# B&R Automation Studio project TD52 (part 11)

#### Sim6CTR.c
```c
/********************************************************************
 * COPYRIGHT -- Bernecker + Rainer Industrie-Elektronik Ges.m.b.H.
 ********************************************************************
 * Program: Sim6CTR
 * File: Sim6CTR.c
 * Author: 105051472
 * Created: Wed Oct 23 10:19:46 2013
 ********************************************************************
 * Implementation of program Sim6CTR
 ********************************************************************
 * Generated with B&R Automation Studio Target for Simulink V4.0
 * (ERT based)
 ********************************************************************/
#include "Sim6CTR.h"
#include "Sim6CTR_private.h"

/*  Defines */

/* Named constants for Chart: '<S1>/Chart' */
#define Sim6CTR_IN_Close_CBP_3u4       ((uint8_T)1U)
#define Sim6CTR_IN_LoadDrop            ((uint8_T)1U)
#define Sim6CTR_IN_Lock_TV             ((uint8_T)1U)
#define Sim6CTR_IN_NO_ACTIVE_CHILD     ((uint8_T)0U)
#define Sim6CTR_IN_Open_CBP_3u4        ((uint8_T)2U)
#define Sim6CTR_IN_Release_TV          ((uint8_T)2U)
#define Sim6CTR_IN_Standard            ((uint8_T)2U)

/*  Data Types */

/**************************** GLOBAL DATA *************************************/
/*  Definitions */

/* Block signals (auto storage) */

/* Block states (auto storage) */

/*  Declarations  */

/***************************** FILE SCOPE DATA ********************************/

/*************************** FUNCTIONS ****************************************/

/* Model step function */
void Sim6CTR_step(struct Sim6CTR* inst)
{
  real_T rtb_Product;
  real_T rtb_Trackingswitch;
  real32_T rtb_Product2_g;
  real32_T rtb_Product1;
  real32_T rtb_Product2_b;
  real32_T rtb_Sum;
  real32_T rtb_Saturation;
  int32_T rtb_Switch1;
  real32_T rtb_Switch_h;
  boolean_T rtb_RelationalOperator2;
  real32_T rtb_Abs;
  real32_T rtb_SumI1;
  real32_T rtb_Saturation_o;
  real32_T rtb_Switch2;
  boolean_T rtb_Compare_e;

  /* S-Function (bur_in): '<Root>/Input10' */
  inst->bur_Sim6CTR_B.Input10 = inst->bInit;

  /* Switch: '<S1>/Switch1' incorporates:
   *  Constant: '<S1>/Constant12'
   *  Constant: '<S1>/Constant3'
   */
  if (inst->bur_Sim6CTR_B.Input10) {
    rtb_Switch1 = 2;
  } else {
    rtb_Switch1 = 3;
  }

  /* End of Switch: '<S1>/Switch1' */

  /* S-Function (bur_in): '<Root>/Input11' */
  inst->bur_Sim6CTR_B.Input11 = inst->Init_Value_CBP;

  /* S-Function (bur_in): '<Root>/Input1' */
  inst->bur_Sim6CTR_B.Input1 = inst->w_set;

  /* Product: '<S7>/Product' */
  rtb_Product = inst->bur_Sim6CTR_B.Input1;

  /* S-Function (bur_in): '<Root>/Input9' */
  inst->bur_Sim6CTR_B.Input9 = inst->x_act;

  /* Sum: '<S7>/Sum' incorporates:
   *  Product: '<S7>/Product1'
   */
  rtb_Product -= (real_T)inst->bur_Sim6CTR_B.Input9;

  /* DeadZone: '<S7>/Deadband' */
  if ((!(rtb_Product > 0.0)) && (rtb_Product >= -0.0)) {
    rtb_Product = 0.0;
  }

  /* End of DeadZone: '<S7>/Deadband' */

  /* Product: '<S7>/Product2' */
  rtb_Product2_g = (real32_T)-rtb_Product;

  /* S-Function (bur_in): '<Root>/Input3' */
  inst->bur_Sim6CTR_B.Input3 = inst->P_CBP;

  /* Product: '<S10>/Product1' incorporates:
   *  Product: '<S7>/Product2'
   */
  rtb_Product1 = (real32_T)-rtb_Product * inst->bur_Sim6CTR_B.Input3;

  /* DiscreteIntegrator: '<S10>/Integrator' */
  rtb_Product2_b = inst->bur_Sim6CTR_DWork.Integrator_DSTATE;

  /* S-Function (bur_in): '<Root>/Input5' */
  inst->bur_Sim6CTR_B.Input5 = inst->D_CBP;

  /* Sum: '<S10>/Sum2' incorporates:
   *  Sum: '<S10>/Sum1'
   */
  rtb_Sum = rtb_Product1 + rtb_Product2_b;

  /* Saturate: '<S10>/Saturation' */
  if (rtb_Sum >= inst->u_max_CBP) {
    rtb_Saturation = inst->u_max_CBP;
  } else if (rtb_Sum <= inst->u_min_CBP) {
    rtb_Saturation = inst->u_min_CBP;
  } else {
    rtb_Saturation = rtb_Sum;
  }

  /* End of Saturate: '<S10>/Saturation' */

  /* MultiPortSwitch: '<S7>/Mode switch' */
  switch (rtb_Switch1) {
   case 1:
    inst->bur_Sim6CTR_B.Modeswitch = inst->bur_Sim6CTR_B.Input11;
    break;

   case 2:
    inst->bur_Sim6CTR_B.Modeswitch = inst->bur_Sim6CTR_B.Input11;
    break;

   default:
    inst->bur_Sim6CTR_B.Modeswitch = rtb_Saturation;
    break;
  }

  /* End of MultiPortSwitch: '<S7>/Mode switch' */

  /* S-Function (bur_out): '<Root>/Output' */
  inst->rPos_CBP = inst->bur_Sim6CTR_B.Modeswitch;

  /* S-Function (bur_in): '<Root>/Input13' */
  inst->bur_Sim6CTR_B.Input13 = inst->rN_act;

  /* S-Function (bur_in): '<Root>/Input12' */
  inst->bur_Sim6CTR_B.Input12 = inst->rN_set;

  /* RelationalOperator: '<S1>/Relational Operator1' incorporates:
   *  Constant: '<S1>/rN_ok_offset'
   *  Sum: '<S1>/Add'
   */
  inst->bur_Sim6CTR_B.RelationalOperator1 = (inst->bur_Sim6CTR_B.Input13 < inst->bur_Sim6CTR_B.Input12 +
    inst->rN_ok_offset);

  /* Switch: '<S9>/Switch' incorporates:
   *  Constant: '<S1>/Cyclic Time'
   *  Constant: '<S9>/Constant4'
   *  Sum: '<S9>/Add'
   *  UnitDelay: '<S6>/Unit Delay2'
   *  UnitDelay: '<S9>/Unit Delay'
   */
  if (inst->bur_Sim6CTR_DWork.UnitDelay2_DSTATE) {
    rtb_Switch_h = 0.0F;
  } else {
    rtb_Switch_h = (real32_T)((real_T)inst->CycleTime + (real_T)
      inst->bur_Sim6CTR_DWork.UnitDelay_DSTATE);
  }

  /* End of Switch: '<S9>/Switch' */

  /* RelationalOperator: '<S6>/Relational Operator2' incorporates:
   *  Constant: '<S1>/Ts_downSampling_speed'
   */
  rtb_RelationalOperator2 = (rtb_Switch_h >= inst->Ts_downSampling_speed);

  /* Switch: '<S6>/Switch' incorporates:
   *  UnitDelay: '<S6>/Unit Delay'
   */
  if (rtb_RelationalOperator2) {
    inst->bur_Sim6CTR_B.Switch = inst->bur_Sim6CTR_B.Input13;
  } else {
    inst->bur_Sim6CTR_B.Switch = inst->bur_Sim6CTR_DWork.UnitDelay_DSTATE_e;
  }

  /* End of Switch: '<S6>/Switch' */

  /* Sum: '<S5>/Diff' incorporates:
   *  UnitDelay: '<S5>/UD'
   */
  inst->bur_Sim6CTR_B.Diff = inst->bur_Sim6CTR_B.Switch - inst->bur_Sim6CTR_DWork.UD_DSTATE;

  /* RelationalOperator: '<S4>/Compare' incorporates:
   *  Constant: '<S4>/Constant'
   */
  inst->bur_Sim6CTR_B.Compare = (inst->bur_Sim6CTR_B.Diff < 0.0F);

  /* Delay: '<S1>/Delay' */
  rtb_Product1 = inst->bur_Sim6CTR_DWork.Delay_DSTATE[0];

  /* S-Function (bur_in): '<Root>/Input2' */
  inst->bur_Sim6CTR_B.Input2 = inst->rP_el;

  /* Sum: '<S1>/Add1' */
  inst->bur_Sim6CTR_B.Add1 = inst->bur_Sim6CTR_B.Input2 - rtb_Product1;

  /* RelationalOperator: '<S1>/Relational Operator' incorporates:
   *  Constant: '<S1>/rP_drop_limit'
   */
  inst->bur_Sim6CTR_B.RelationalOperator = (inst->bur_Sim6CTR_B.Add1 < inst->rP_drop_limit);

  /* Chart: '<S1>/Chart' incorporates:
   *  Constant: '<S1>/rP_el_LockTV'
   *  MinMax: '<S1>/MinMax'
   *  UnitDelay: '<S1>/Unit Delay'
   */
  /* Gateway: Island Controller/Chart */
  /* During: Island Controller/Chart */
  if (inst->bur_Sim6CTR_DWork.is_active_c1_Sim6CTR == 0U) {
    /* Entry: Island Controller/Chart */
    inst->bur_Sim6CTR_DWork.is_active_c1_Sim6CTR = 1U;

    /* Entry Internal: Island Controller/Chart */
    /* Transition: '<S3>:12' */
    inst->bur_Sim6CTR_DWork.is_c1_Sim6CTR = Sim6CTR_IN_Standard;

    /* Entry 'Standard': '<S3>:7' */
    inst->bur_Sim6CTR_B.bLoadDrop = FALSE;
    inst->bur_Sim6CTR_B.Open4CBP = FALSE;

    /* Entry Internal 'Standard': '<S3>:7' */
    /* Transition: '<S3>:16' */
    inst->bur_Sim6CTR_DWork.is_Standard = Sim6CTR_IN_Release_TV;

    /* Entry 'Release_TV': '<S3>:15' */
    inst->bur_Sim6CTR_B.Lock_TV = FALSE;
    inst->bur_Sim6CTR_B.Control_State = 11;
  } else if (inst->bur_Sim6CTR_DWork.is_c1_Sim6CTR == Sim6CTR_IN_LoadDrop) {
    /* During 'LoadDrop': '<S3>:10' */
    if (inst->bur_Sim6CTR_B.RelationalOperator1 && inst->bur_Sim6CTR_B.Compare) {
      /* Transition: '<S3>:25' */
      /* Exit Internal 'LoadDrop': '<S3>:10' */
      inst->bur_Sim6CTR_DWork.is_LoadDrop = Sim6CTR_IN_NO_ACTIVE_CHILD;
      inst->bur_Sim6CTR_DWork.is_c1_Sim6CTR = Sim6CTR_IN_Standard;

      /* Entry 'Standard': '<S3>:7' */
      inst->bur_Sim6CTR_B.bLoadDrop = FALSE;
      inst->bur_Sim6CTR_B.Open4CBP = FALSE;

      /* Entry Internal 'Standard': '<S3>:7' */
      /* Transition: '<S3>:16' */
      inst->bur_Sim6CTR_DWork.is_Standard = Sim6CTR_IN_Release_TV;

      /* Entry 'Release_TV': '<S3>:15' */
      inst->bur_Sim6CTR_B.Lock_TV = FALSE;
      inst->bur_Sim6CTR_B.Control_State = 11;
    } else {
      switch (inst->bur_Sim6CTR_DWork.is_LoadDrop) {
       case Sim6CTR_IN_Close_CBP_3u4:
        break;

       default:
        /* During 'Open_CBP_3u4': '<S3>:29' */
        if (inst->bur_Sim6CTR_B.Compare) {
          /* Transition: '<S3>:32' */
          inst->bur_Sim6CTR_DWork.is_LoadDrop = Sim6CTR_IN_Close_CBP_3u4;

          /* Entry 'Close_CBP_3u4': '<S3>:31' */
          inst->bur_Sim6CTR_B.Open4CBP = FALSE;
          inst->bur_Sim6CTR_B.Control_State = 22;
        }
        break;
      }
    }
  } else {
    /* During 'Standard': '<S3>:7' */
    if (inst->bur_Sim6CTR_B.RelationalOperator) {
      /* Transition: '<S3>:23' */
      /* Exit Internal 'Standard': '<S3>:7' */
      inst->bur_Sim6CTR_DWork.is_Standard = Sim6CTR_IN_NO_ACTIVE_CHILD;
      inst->bur_Sim6CTR_DWork.is_c1_Sim6CTR = Sim6CTR_IN_LoadDrop;

      /* Entry 'LoadDrop': '<S3>:10' */
      inst->bur_Sim6CTR_B.Lock_TV = FALSE;
      inst->bur_Sim6CTR_B.bLoadDrop = TRUE;

      /* Entry Internal 'LoadDrop': '<S3>:10' */
      /* Transition: '<S3>:30' */
      inst->bur_Sim6CTR_DWork.is_LoadDrop = Sim6CTR_IN_Open_CBP_3u4;

      /* Entry 'Open_CBP_3u4': '<S3>:29' */
      inst->bur_Sim6CTR_B.Open4CBP = TRUE;
      inst->bur_Sim6CTR_B.Control_State = 21;
    } else if (inst->bur_Sim6CTR_DWork.is_Standard == Sim6CTR_IN_Lock_TV) {
      /* MinMax: '<S1>/MinMax' incorporates:
       *  Constant: '<S1>/rP_el_LockTV'
       *  Constant: '<S1>/rP_el_ReleaseTV'
       */
      /* During 'Lock_TV': '<S3>:9' */
      if (inst->rP_el_LockTV <= inst->rP_el_ReleaseTV) {
        rtb_Product = inst->rP_el_LockTV;
      } else {
        rtb_Product = inst->rP_el_ReleaseTV;
      }

      if ((real_T)inst->bur_Sim6CTR_B.Input2 < rtb_Product) {
        /* Transition: '<S3>:20' */
        inst->bur_Sim6CTR_DWork.is_Standard = Sim6CTR_IN_Release_TV;

        /* Entry 'Release_TV': '<S3>:15' */
        inst->bur_Sim6CTR_B.Lock_TV = FALSE;
        inst->bur_Sim6CTR_B.Control_State = 11;
      }
    } else {
      /* During 'Release_TV': '<S3>:15' */
      if ((inst->bur_Sim6CTR_B.Input2 > inst->rP_el_LockTV) && (inst->bur_Sim6CTR_DWork.UnitDelay_DSTATE_n
           > 72.0F)) {
        /* Transition: '<S3>:19' */
        inst->bur_Sim6CTR_DWork.is_Standard = Sim6CTR_IN_Lock_TV;

        /* Entry 'Lock_TV': '<S3>:9' */
        inst->bur_Sim6CTR_B.Lock_TV = TRUE;
        inst->bur_Sim6CTR_B.Control_State = 12;
      }
    }
  }

  /* End of Chart: '<S1>/Chart' */

  /* Switch: '<S1>/Switch' incorporates:
   *  Constant: '<S1>/Constant2'
   *  Constant: '<S1>/Constant31'
   *  Logic: '<S1>/Logical Operator'
   */
  if (inst->bur_Sim6CTR_B.Input10 || inst->bur_Sim6CTR_B.Lock_TV) {
    rtb_Product = 2.0;
  } else {
    rtb_Product = 3.0;
  }

  /* End of Switch: '<S1>/Switch' */

  /* S-Function (bur_in): '<Root>/Input14' */
  inst->bur_Sim6CTR_B.Input14 = inst->Init_Value_TV;

  /* Switch: '<S1>/Switch2' incorporates:
   *  Constant: '<S1>/u_man_TV'
   */
  if (inst->bur_Sim6CTR_B.Input10) {
    rtb_Switch2 = inst->bur_Sim6CTR_B.Input14;
  } else {
    rtb_Switch2 = inst->u_man_TV;
  }

  /* End of Switch: '<S1>/Switch2' */

  /* Sum: '<S8>/Sum' incorporates:
   *  Product: '<S8>/Product'
   *  Product: '<S8>/Product1'
   */
  rtb_Trackingswitch = (real_T)inst->bur_Sim6CTR_B.Input1 - (real_T)inst->bur_Sim6CTR_B.Input9;

  /* DeadZone: '<S8>/Deadband' */
  if ((!(rtb_Trackingswitch > 0.0)) && (rtb_Trackingswitch >= -0.0)) {
    rtb_Trackingswitch = 0.0;
  }

  /* End of DeadZone: '<S8>/Deadband' */

  /* Product: '<S8>/Product2' */
  rtb_Product2_b = (real32_T)rtb_Trackingswitch;

  /* S-Function (bur_in): '<Root>/Input6' */
  inst->bur_Sim6CTR_B.Input6 = inst->P_TV;

  /* Product: '<S13>/Product1' incorporates:
   *  Product: '<S8>/Product2'
   */
  rtb_Product1 = (real32_T)rtb_Trackingswitch * inst->bur_Sim6CTR_B.Input6;

  /* DiscreteIntegrator: '<S13>/Integrator' */
  rtb_Abs = inst->bur_Sim6CTR_DWork.Integrator_DSTATE_i;

  /* S-Function (bur_in): '<Root>/Input8' */
  inst->bur_Sim6CTR_B.Input8 = inst->D_TV;

  /* Sum: '<S13>/Sum2' incorporates:
   *  Sum: '<S13>/Sum1'
   */
  rtb_SumI1 = rtb_Product1 + rtb_Abs;

  /* Saturate: '<S13>/Saturation' */
  if (rtb_SumI1 >= inst->u_max_TV) {
    rtb_Saturation_o = inst->u_max_TV;
  } else if (rtb_SumI1 <= inst->u_min_TV) {
    rtb_Saturation_o = inst->u_min_TV;
  } else {
    rtb_Saturation_o = rtb_SumI1;
  }

  /* End of Saturate: '<S13>/Saturation' */

  /* MultiPortSwitch: '<S8>/Mode switch' */
  switch ((int32_T)rtb_Product) {
   case 1:
    inst->bur_Sim6CTR_B.Modeswitch_a = rtb_Switch2;
    break;

   case 2:
    inst->bur_Sim6CTR_B.Modeswitch_a = rtb_Switch2;
    break;

   default:
    inst->bur_Sim6CTR_B.Modeswitch_a = rtb_Saturation_o;
    break;
  }

  /* End of MultiPortSwitch: '<S8>/Mode switch' */

  /* S-Function (bur_out): '<Root>/Output1' */
  inst->rPos_TV = inst->bur_Sim6CTR_B.Modeswitch_a;

  /* S-Function (bur_out): '<Root>/Output10' */
  inst->rN_act_Diff = inst->bur_Sim6CTR_B.Diff;

  /* S-Function (bur_out): '<Root>/Output11' */
  inst->bOpen4CBP = inst->bur_Sim6CTR_B.Open4CBP;

  /* S-Function (bur_out): '<Root>/Output2' */
  inst->bLoadDrop = inst->bur_Sim6CTR_B.bLoadDrop;

  /* S-Function (bur_out): '<Root>/Output3' */
  inst->Control_State = inst->bur_Sim6CTR_B.Control_State;

  /* S-Function (bur_out): '<Root>/Output4' */
  inst->bLock_TV = inst->bur_Sim6CTR_B.Lock_TV;

  /* S-Function (bur_out): '<Root>/Output5' */
  inst->bN_ok = inst->bur_Sim6CTR_B.RelationalOperator1;

  /* S-Function (bur_out): '<Root>/Output6' */
  inst->bN_rate_neg = inst->bur_Sim6CTR_B.Compare;

  /* S-Function (bur_out): '<Root>/Output7' */
  inst->bP_drop = inst->bur_Sim6CTR_B.RelationalOperator;

  /* S-Function (bur_out): '<Root>/Output8' */
  inst->rP_grad = inst->bur_Sim6CTR_B.Add1;

  /* S-Function (bur_out): '<Root>/Output9' */
  inst->rN_act_DS = inst->bur_Sim6CTR_B.Switch;

  /* S-Function (bur_in): '<Root>/Input4' */
  inst->bur_Sim6CTR_B.Input4 = inst->I_CBP;

  /* S-Function (bur_in): '<Root>/Input7' */
  inst->bur_Sim6CTR_B.Input7 = inst->I_TV;

  /* Sum: '<S11>/Sum' */
  rtb_Sum = rtb_Saturation - rtb_Sum;

  /* MultiPortSwitch: '<S7>/Tracking switch' incorporates:
   *  Constant: '<S7>/Constant'
   *  Constant: '<S7>/Constant1'
   */
  switch (rtb_Switch1) {
   case 1:
    rtb_Trackingswitch = 0.0;
    break;

   case 2:
    rtb_Trackingswitch = 1.0;
    break;

   default:
    rtb_Trackingswitch = 0.0;
    break;
  }

  /* End of MultiPortSwitch: '<S7>/Tracking switch' */

  /* Sum: '<S10>/SumI1' incorporates:
   *  Product: '<S10>/Product'
   *  Product: '<S10>/Product2'
   *  Sum: '<S10>/SumI3'
   */
  rtb_Abs = (real32_T)((real_T)(inst->bur_Sim6CTR_B.Input11 - rtb_Saturation) *
                       rtb_Trackingswitch) + rtb_Product2_g * inst->bur_Sim6CTR_B.Input4;

  /* Signum: '<S11>/SignPreSat' */
  if (rtb_Sum < 0.0F) {
    rtb_Product2_g = -1.0F;
  } else if (rtb_Sum > 0.0F) {
    rtb_Product2_g = 1.0F;
  } else {
    rtb_Product2_g = rtb_Sum;
  }

  /* Signum: '<S11>/SignPreIntegrator' */
  if (rtb_Abs < 0.0F) {
    rtb_Saturation = -1.0F;
  } else if (rtb_Abs > 0.0F) {
    rtb_Saturation = 1.0F;
  } else {
    rtb_Saturation = rtb_Abs;
  }

  /* Switch: '<S10>/Switch' incorporates:
   *  Abs: '<S11>/Abs'
   *  Constant: '<S10>/Constant4'
   *  Constant: '<S12>/Constant'
   *  Logic: '<S11>/AND'
   *  RelationalOperator: '<S11>/Equal'
   *  RelationalOperator: '<S12>/Compare'
   *  Signum: '<S11>/SignPreIntegrator'
   *  Signum: '<S11>/SignPreSat'
   */
  if (((real32_T)fabs(rtb_Sum) > 0.1F) && (rtb_Product2_g != rtb_Saturation)) {
    rtb_Abs = 0.0F;
  }

  /* End of Switch: '<S10>/Switch' */

  /* Sum: '<S14>/Sum' */
  rtb_SumI1 = rtb_Saturation_o - rtb_SumI1;

  /* RelationalOperator: '<S15>/Compare' incorporates:
   *  Abs: '<S14>/Abs'
   *  Constant: '<S15>/Constant'
   */
  rtb_Compare_e = ((real32_T)fabs(rtb_SumI1) > 0.1F);

  /* Signum: '<S14>/SignPreSat' */
  if (rtb_SumI1 < 0.0F) {
    rtb_Product1 = -1.0F;
  } else if (rtb_SumI1 > 0.0F) {
    rtb_Product1 = 1.0F;
  } else {
    rtb_Product1 = rtb_SumI1;
  }

  /* End of Signum: '<S14>/SignPreSat' */

  /* MultiPortSwitch: '<S8>/Tracking switch' incorporates:
   *  Constant: '<S8>/Constant'
   *  Constant: '<S8>/Constant1'
   */
  switch ((int32_T)rtb_Product) {
   case 1:
    rtb_Trackingswitch = 0.0;
    break;

   case 2:
    rtb_Trackingswitch = 1.0;
    break;

   default:
    rtb_Trackingswitch = 0.0;
    break;
  }

  /* End of MultiPortSwitch: '<S8>/Tracking switch' */

  /* Sum: '<S13>/SumI1' incorporates:
   *  Product: '<S13>/Product'
   *  Product: '<S13>/Product2'
   *  Sum: '<S13>/SumI3'
   */
  rtb_SumI1 = (real32_T)((real_T)(rtb_Switch2 - rtb_Saturation_o) *
    rtb_Trackingswitch) + rtb_Product2_b * inst->bur_Sim6CTR_B.Input7;

  /* Signum: '<S14>/SignPreIntegrator' */
  if (rtb_SumI1 < 0.0F) {
    rtb_Product2_g = -1.0F;
  } else if (rtb_SumI1 > 0.0F) {
    rtb_Product2_g = 1.0F;
  } else {
    rtb_Product2_g = rtb_SumI1;
  }

  /* Switch: '<S13>/Switch' incorporates:
   *  Constant: '<S13>/Constant4'
   *  Logic: '<S14>/AND'
   *  RelationalOperator: '<S14>/Equal'
   *  Signum: '<S14>/SignPreIntegrator'
   */
  if (rtb_Compare_e && (rtb_Product1 != rtb_Product2_g)) {
    rtb_Product1 = 0.0F;
  } else {
    rtb_Product1 = rtb_SumI1;
  }

  /* End of Switch: '<S13>/Switch' */

  /* Update for DiscreteIntegrator: '<S10>/Integrator' */
  inst->bur_Sim6CTR_DWork.Integrator_DSTATE += 0.01F * rtb_Abs;

  /* Update for UnitDelay: '<S6>/Unit Delay2' */
  inst->bur_Sim6CTR_DWork.UnitDelay2_DSTATE = rtb_RelationalOperator2;

  /* Update for UnitDelay: '<S9>/Unit Delay' */
  inst->bur_Sim6CTR_DWork.UnitDelay_DSTATE = rtb_Switch_h;

  /* Update for UnitDelay: '<S6>/Unit Delay' */
  inst->bur_Sim6CTR_DWork.UnitDelay_DSTATE_e = inst->bur_Sim6CTR_B.Switch;

  /* Update for UnitDelay: '<S5>/UD' */
  inst->bur_Sim6CTR_DWork.UD_DSTATE = inst->bur_Sim6CTR_B.Switch;

  /* Update for Delay: '<S1>/Delay' */
  for (rtb_Switch1 = 0; rtb_Switch1 < 9; rtb_Switch1++) {
    inst->bur_Sim6CTR_DWork.Delay_DSTATE[rtb_Switch1] =
      inst->bur_Sim6CTR_DWork.Delay_DSTATE[rtb_Switch1 + 1];
  }

  inst->bur_Sim6CTR_DWork.Delay_DSTATE[9] = inst->bur_Sim6CTR_B.Input2;

  /* End of Update for Delay: '<S1>/Delay' */

  /* Update for UnitDelay: '<S1>/Unit Delay' */
  inst->bur_Sim6CTR_DWork.UnitDelay_DSTATE_n = inst->bur_Sim6CTR_B.Modeswitch_a;

  /* Update for DiscreteIntegrator: '<S13>/Integrator' */
  inst->bur_Sim6CTR_DWork.Integrator_DSTATE_i += 0.01F * rtb_Product1;
}

/* Model initialize function */
void Sim6CTR_initialize(struct Sim6CTR* inst)
{
  /* InitializeConditions for Chart: '<S1>/Chart' */
  inst->bur_Sim6CTR_B.Control_State = 0;
  inst->bur_Sim6CTR_B.Lock_TV = FALSE;
  inst->bur_Sim6CTR_B.bLoadDrop = FALSE;
  inst->bur_Sim6CTR_B.Open4CBP = FALSE;
}

/* Model terminate function */
void Sim6CTR_terminate(struct Sim6CTR* inst)
{
  /* (no terminate code required) */
}

/*======================== TOOL VERSION INFORMATION ==========================*
 * MATLAB 8.0 (R2012b)20-Jul-2012                                             *
 * Simulink 8.0 (R2012b)20-Jul-2012                                           *
 * Simulink Coder 8.3 (R2012b)20-Jul-2012                                     *
 * Embedded Coder 6.3 (R2012b)20-Jul-2012                                     *
 * Stateflow 8.0 (R2012b)20-Jul-2012                                          *
 *============================================================================*/

/*======================= LICENSE IN USE INFORMATION =========================*
 * control_toolbox                                                            *
 * identification_toolbox                                                     *
 * matlab                                                                     *
 * matlab_coder                                                               *
 * real-time_workshop                                                         *
 * rtw_embedded_coder                                                         *
 * simulink                                                                   *
 * stateflow                                                                  *
 *============================================================================*/
```

#### main.c
```c
/********************************************************************
 * COPYRIGHT -- Bernecker + Rainer Industrie-Elektronik Ges.m.b.H.
 ********************************************************************
 * Program: Sim6CTR
 * File: main.c
 * Author: 105051472
 * Created: Wed Oct 23 10:19:46 2013
 ********************************************************************
 * Implementation of program Sim6CTR
 ********************************************************************
 * Generated with B&R Automation Studio Target for Simulink V4.0
 * (ERT based)
 ********************************************************************/
#include <bur/plctypes.h>
#include "Sim6CTR.h"
#include "rtwtypes.h"

BOOL bur_firsttime = TRUE;

/*  Defines */
#define SS_TERMINATE 4
#define SS_OUTPUT 3
#define SS_INITIALIZE 2

/*  Data Types */

/**************************** GLOBAL DATA *************************************/
/*  Definitions */

/*  Declarations  */

/***************************** FILE SCOPE DATA ********************************/

/*************************** FUNCTIONS ****************************************/
#ifdef __cplusplus

unsigned long bur_heap_size = 65535;

#endif

void Sim6CTR(struct Sim6CTR* inst)
{
  switch (inst->ssMethodType)
  {
   case SS_INITIALIZE:
    /* call model initialize function */
    Sim6CTR_initialize(inst);
    break;

   case SS_OUTPUT:
    /* call model step function */
    Sim6CTR_step(inst);

    break;

   case SS_TERMINATE:
    /* call model terminate function */
    Sim6CTR_terminate(inst);
    break;
  }
}

/*****************************************************************************
   Function block sample time: 0.01s
 *****************************************************************************/

/*****************************************************************************
   B&R Automation Studio Target for Simulink Version: A4.0.48 (27-Jun-2013)
 *****************************************************************************/

/*======================== TOOL VERSION INFORMATION ==========================*
 * MATLAB 8.0 (R2012b)20-Jul-2012                                             *
 * Simulink 8.0 (R2012b)20-Jul-2012                                           *
 * Simulink Coder 8.3 (R2012b)20-Jul-2012                                     *
 * Embedded Coder 6.3 (R2012b)20-Jul-2012                                     *
 * Stateflow 8.0 (R2012b)20-Jul-2012                                          *
 *============================================================================*/

/*======================= LICENSE IN USE INFORMATION =========================*
 * control_toolbox                                                            *
 * identification_toolbox                                                     *
 * matlab                                                                     *
 * matlab_coder                                                               *
 * real-time_workshop                                                         *
 * rtw_embedded_coder                                                         *
 * simulink                                                                   *
 * stateflow                                                                  *
 *============================================================================*/
```

#### lib_properties.txt
```
For manual assignment to hardware configuration please
add the following additional include directories:

\Logical\MATLAB_includes\R2012b\

And the following additional build options:

-lm -D MODEL=Sim6CTR -D NUMST=1 -D NCSTATES=0 -D HAVESTDIO -D ONESTEPFCN=1 -D TERMFCN=1 -D MAT_FILE=0 -D MULTI_INSTANCE_CODE=0 -D INTEGER_CODE=0 -D MT=0 -D CLASSIC_INTERFACE=0 -D TID01EQ=0
```

### Library Logical/Libraries/lLamCorr (ANSIC)

#### lLamCorr.fun
```iecst
FUNCTION_BLOCK lLamCorr
  VAR_INPUT
    ssMethodType: SINT;
  END_VAR  VAR_INPUT
        rN_Set : REAL := 1500.0000000000; (*speed set value [rpm]*)
  END_VAR
  VAR_INPUT
        rP_Nom : REAL := 4400.0000000000; (*nominal power [KW]*)
  END_VAR
  VAR_INPUT
        rN_Delta_Lim : REAL := 0.0099999998; (*delta speed limit when engine speed is recovered, normed*)
  END_VAR
  VAR_INPUT
        rP_Rot_Norm_Lam_Trig : REAL := 0.0199999996; (*rotational power trigger value for lambda adaption, normed*)
  END_VAR
  VAR_INPUT
        rP_Rot_Norm_Lambda_Gain : REAL := 1.0000000000; (*gain value to convert nomed rotational power to delta lambda value for lambda adaption*)
  END_VAR
  VAR_INPUT
        rLam_OffsLimit_pos : REAL; (*pos limitation of dynamic lambda offset*)
  END_VAR
  VAR_INPUT
        rLam_Ramp_Grad : REAL := 0.2500000000; (*neg limitation of dynamic lambda offset*)
  END_VAR
  VAR_INPUT
        bLambda_Corr_Enable : BOOL := FALSE; (*enable function of lambda correction*)
  END_VAR
  VAR_INPUT
        rP_Rot : REAL; (*rotational power*)
  END_VAR
  VAR_INPUT
        rN_Eng : REAL; (*engine speed [rpm]*)
  END_VAR
  VAR_INPUT
        rLam_OffsLimit_Neg : REAL; (*engine speed [rpm]*)
  END_VAR
  VAR_OUTPUT
        rLambda_Corr : REAL; (*Lambda adaption value*)
  END_VAR
  VAR_OUTPUT
        bLambda_Freeze : BOOL := FALSE; (*Lambda adaption value*)
  END_VAR
  VAR_OUTPUT
        rP_Rot_Max : REAL; (*maximum value for rotational power, used for calibration*)
  END_VAR
  VAR_OUTPUT
        bN_Delta_Act : BOOL := FALSE; (*Debug Output*)
  END_VAR
  VAR_OUTPUT
        bP_Rot_Lambda_Act : BOOL := FALSE; (*Debug Output*)
  END_VAR
  VAR_OUTPUT
        bN_Delta_Neg : BOOL := FALSE; (*Debug Output*)
  END_VAR
	VAR
		bur_BlockIO_LambdaAdp : BlockIO_LambdaAdp;
	END_VAR
	VAR
		bur_D_Work_LambdaAdp : D_Work_LambdaAdp;
	END_VAR
END_FUNCTION_BLOCK
```

#### lLamCorr.typ
```iecst
TYPE

END_TYPE
TYPE
BlockIO_LambdaAdp : STRUCT
	Input1 : REAL;
	Input2 : REAL;
	Input3 : REAL;
	DifferenceInputs2 : REAL;
	MinMax : REAL;
	Input4 : BOOL;
	RelationalOperator2 : BOOL;
	RelationalOperator : BOOL;
	RelationalOperator1 : BOOL;
	bLambda_Corr_Act : BOOL;
END_STRUCT;
D_Work_LambdaAdp : STRUCT
	DelayInput2_DSTATE : REAL;
	UnitDelay_DSTATE : REAL;
	is_active_c1_LambdaAdp : USINT;
	is_c1_LambdaAdp : USINT;
	MAX_MODE : BOOL;
END_STRUCT;
END_TYPE
```

#### LambdaAdp.h
```c
/********************************************************************
 * COPYRIGHT -- Bernecker + Rainer Industrie-Elektronik Ges.m.b.H.
 ********************************************************************
 * Program: LambdaAdp
 * File: LambdaAdp.h
 * Author: 105051472
 * Created: Wed Oct 29 12:06:16 2014
 ********************************************************************
 * Header for program LambdaAdp
 ********************************************************************
 * Generated with B&R Automation Studio Target for Simulink V4.2
 * (ERT based)
 ********************************************************************/

#ifndef RTW_HEADER_LambdaAdp_h_
#define RTW_HEADER_LambdaAdp_h_
#ifndef LambdaAdp_COMMON_INCLUDES_
# define LambdaAdp_COMMON_INCLUDES_
#include "rtwtypes.h"
#endif                                 /* LambdaAdp_COMMON_INCLUDES_ */

#include "LambdaAdp_types.h"
#include "lLamCorr.h"

/* Macros for accessing real-time model data structure */
#ifndef rtmGetErrorStatus
# define rtmGetErrorStatus(rtm)        ((void*) 0)
#endif

#ifndef rtmSetErrorStatus
# define rtmSetErrorStatus(rtm, val)   ((void) 0)
#endif

#ifndef rtmGetStopRequested
# define rtmGetStopRequested(rtm)      ((void*) 0)
#endif

#ifndef MIN
#define MIN(a,b)                       ((a) < (b) ? (a) : (b))
#endif

#ifndef MAX
#define MAX(a,b)                       ((a) > (b) ? (a) : (b))
#endif

/* Block signals (auto storage) */

/* Block states (auto storage) for system '<Root>' */

/* Block signals (auto storage) */
extern BlockIO_LambdaAdp LambdaAdp_B;

/* Block states (auto storage) */
extern D_Work_LambdaAdp LambdaAdp_DWork;

/* Model entry point functions */
extern void LambdaAdp_initialize(struct lLamCorr* inst);
extern void LambdaAdp_step(struct lLamCorr* inst);
extern void LambdaAdp_terminate(struct lLamCorr* inst);

/*-
 * The generated code includes comments that allow you to trace directly
 * back to the appropriate location in the model.  The basic format
 * is <system>/block_name, where system is the system number (uniquely
 * assigned by Simulink) and block_name is the name of the block.
 *
 * Use the MATLAB hilite_system command to trace the generated code back
 * to the model.  For example,
 *
 * hilite_system('<S3>')    - opens system 3
 * hilite_system('<S3>/Kp') - opens and selects block Kp which resides in S3
 *
 * Here is the system hierarchy for this model
 *
 * '<Root>' : 'LambdaAdp'
 * '<S1>'   : 'LambdaAdp/LambdaAdaption'
 * '<S2>'   : 'LambdaAdp/LambdaAdaption/Lambda_Active'
 * '<S3>'   : 'LambdaAdp/LambdaAdaption/MAX'
 * '<S4>'   : 'LambdaAdp/LambdaAdaption/Rate Limiter Dynamic'
 * '<S5>'   : 'LambdaAdp/LambdaAdaption/Saturation Dynamic'
 * '<S6>'   : 'LambdaAdp/LambdaAdaption/Rate Limiter Dynamic/Saturation Dynamic'
 */
#endif                                 /* RTW_HEADER_LambdaAdp_h_ */
```

#### LambdaAdp_private.h
```c
/********************************************************************
 * COPYRIGHT -- Bernecker + Rainer Industrie-Elektronik Ges.m.b.H.
 ********************************************************************
 * Program: LambdaAdp
 * File: LambdaAdp_private.h
 * Author: 105051472
 * Created: Wed Oct 29 12:06:16 2014
 ********************************************************************
 * Header for program LambdaAdp
 ********************************************************************
 * Generated with B&R Automation Studio Target for Simulink V4.2
 * (ERT based)
 ********************************************************************/

#ifndef RTW_HEADER_LambdaAdp_private_h_
#define RTW_HEADER_LambdaAdp_private_h_
#include "rtwtypes.h"
#include <bur/plctypes.h>
#ifndef __RTWTYPES_H__
#error This file requires rtwtypes.h to be included
#else
#ifdef TMWTYPES_PREVIOUSLY_INCLUDED
#error This file requires rtwtypes.h to be included before tmwtypes.h
#else

/* Check for inclusion of an incorrect version of rtwtypes.h */
#ifndef RTWTYPES_ID_C08S16I32L32N32F1
#error This code was generated with a different "rtwtypes.h" than the file included
#endif                                 /* RTWTYPES_ID_C08S16I32L32N32F1 */
#endif                                 /* TMWTYPES_PREVIOUSLY_INCLUDED */
#endif                                 /* __RTWTYPES_H__ */

#ifndef MIN
#define MIN(a,b)                       ((a) < (b) ? (a) : (b))
#endif

#ifndef MAX
#define MAX(a,b)                       ((a) > (b) ? (a) : (b))
#endif

/* Imported (extern) block parameters */
extern real32_T rLam_OffsLimit_pos;    /* Variable: rLam_OffsLimit_pos
                                        * Referenced by: '<S1>/rLam_OffsLimit_pos'
                                        */
extern real32_T rLam_Ramp_Grad;        /* Variable: rLam_Ramp_Grad
                                        * Referenced by: '<S1>/rLam_Ramp_Grad'
                                        */
extern real32_T rN_Delta_Lim;          /* Variable: rN_Delta_Lim
                                        * Referenced by: '<S1>/rN_Delta_Lim'
                                        */
extern real32_T rN_Set;                /* Variable: rN_Set
                                        * Referenced by: '<S1>/rN_Set'
                                        */
extern real32_T rP_Nom;                /* Variable: rP_Nom
                                        * Referenced by: '<S1>/rP_Nom'
                                        */
extern real32_T rP_Rot_Norm_Lam_Trig;  /* Variable: rP_Rot_Norm_Lam_Trig
                                        * Referenced by: '<S1>/rP_Rot_Norm_Lam_Trig'
                                        */
extern real32_T rP_Rot_Norm_Lambda_Gain;/* Variable: rP_Rot_Norm_Lambda_Gain
                                         * Referenced by: '<S1>/rP_Rot_Norm_Lambda_Gain'
                                         */

#endif                                 /* RTW_HEADER_LambdaAdp_private_h_ */
```

#### LambdaAdp_types.h
```c
/********************************************************************
 * COPYRIGHT -- Bernecker + Rainer Industrie-Elektronik Ges.m.b.H.
 ********************************************************************
 * Program: LambdaAdp
 * File: LambdaAdp_types.h
 * Author: 105051472
 * Created: Wed Oct 29 12:06:16 2014
 ********************************************************************
 * Header for program LambdaAdp
 ********************************************************************
 * Generated with B&R Automation Studio Target for Simulink V4.2
 * (ERT based)
 ********************************************************************/

#ifndef RTW_HEADER_LambdaAdp_types_h_
#define RTW_HEADER_LambdaAdp_types_h_
#ifndef MIN
#define MIN(a,b)                       ((a) < (b) ? (a) : (b))
#endif

#ifndef MAX
#define MAX(a,b)                       ((a) > (b) ? (a) : (b))
#endif
#endif                                 /* RTW_HEADER_LambdaAdp_types_h_ */
```

#### rtwtypes.h
```c
/********************************************************************
 * COPYRIGHT -- Bernecker + Rainer Industrie-Elektronik Ges.m.b.H.
 ********************************************************************
 * Program: LambdaAdp
 * File: rtwtypes.h
 * Author: 105051472
 * Created: Wed Oct 29 12:06:16 2014
 ********************************************************************
 * Header for program LambdaAdp
 ********************************************************************
 * Generated with B&R Automation Studio Target for Simulink V4.2
 * (ERT based)
 ********************************************************************/

#ifndef __RTWTYPES_H__
#define __RTWTYPES_H__
#ifndef TRUE
# define TRUE                          (1U)
#endif

#ifndef FALSE
# define FALSE                         (0U)
#endif

#ifndef __TMWTYPES__
#define __TMWTYPES__
#include <limits.h>

/*=======================================================================*
 * Target hardware information
 *   Device type: Intel->x86/Pentium
 *   Number of bits:     char:   8    short:   16    int:  32
 *                       long:  32
 *                       native word size:  32
 *   Byte ordering: LittleEndian
 *   Signed integer division rounds to: Zero
 *   Shift right on a signed integer as arithmetic shift: on
 *=======================================================================*/

/*=======================================================================*
 * Fixed width word size data types:                                     *
 *   int8_T, int16_T, int32_T     - signed 8, 16, or 32 bit integers     *
 *   uint8_T, uint16_T, uint32_T  - unsigned 8, 16, or 32 bit integers   *
 *   real32_T, real64_T           - 32 and 64 bit floating point numbers *
 *=======================================================================*/
typedef signed char int8_T;
typedef unsigned char uint8_T;
typedef short int16_T;
typedef unsigned short uint16_T;
typedef int int32_T;
typedef unsigned int uint32_T;
typedef float real32_T;
typedef double real64_T;

/*===========================================================================*
 * Generic type definitions: real_T, time_T, boolean_T, int_T, uint_T,       *
 *                           ulong_T, char_T and byte_T.                     *
 *===========================================================================*/
typedef double real_T;
typedef double time_T;
typedef unsigned char boolean_T;
typedef long int int_T;
typedef unsigned int uint_T;
typedef unsigned long ulong_T;
typedef char char_T;
typedef unsigned char uchar_T;
typedef char_T byte_T;

/*=======================================================================*
 * Min and Max:                                                          *
 *   int8_T, int16_T, int32_T     - signed 8, 16, or 32 bit integers     *
 *   uint8_T, uint16_T, uint32_T  - unsigned 8, 16, or 32 bit integers   *
 *=======================================================================*/
#define MAX_int8_T                     ((int8_T)(127))
#define MIN_int8_T                     ((int8_T)(-128))
#define MAX_uint8_T                    ((uint8_T)(255U))
#define MIN_uint8_T                    ((uint8_T)(0U))
#define MAX_int16_T                    ((int16_T)(32767))
#define MIN_int16_T                    ((int16_T)(-32768))
#define MAX_uint16_T                   ((uint16_T)(65535U))
#define MIN_uint16_T                   ((uint16_T)(0U))
#define MAX_int32_T                    ((int32_T)(2147483647))
#define MIN_int32_T                    ((int32_T)(-2147483647-1))
#define MAX_uint32_T                   ((uint32_T)(0xFFFFFFFFU))
#define MIN_uint32_T                   ((uint32_T)(0U))

/* Logical type definitions */
#if (!defined(__cplusplus)) && (!defined(__true_false_are_keywords))
#  ifndef false
#   define false                       (0U)
#  endif

#  ifndef true
#   define true                        (1U)
#  endif
#endif

/*
 * Simulink Coder assumes the code is compiled on a target using a 2's complement representation
 * for signed integer values.
 */
#if ((SCHAR_MIN + 1) != -SCHAR_MAX)
#error "This code must be compiled using a 2's complement representation for signed integer values"
#endif

/* This ID is used to detect inclusion of an incompatible rtwtypes.h */
#define RTWTYPES_ID_C08S16I32L32N32F1
#else                                  /* __TMWTYPES__ */
#define TMWTYPES_PREVIOUSLY_INCLUDED
#endif                                 /* __TMWTYPES__ */

/* Block D-Work pointer type */
typedef void * pointer_T;

/* Simulink specific types */
#ifndef __SIMSTRUC_TYPES_H__
#define __SIMSTRUC_TYPES_H__

/* Trigger directions: falling, either, and rising */
typedef enum {
  FALLING_ZERO_CROSSING = -1,
  ANY_ZERO_CROSSING = 0,
  RISING_ZERO_CROSSING = 1
} ZCDirection;

/* Previous state of a trigger signal */
typedef uint8_T ZCSigState;

/* Initial value of a trigger zero crossing signal */
#define UNINITIALIZED_ZCSIG            0x03U
#define NEG_ZCSIG                      0x02U
#define POS_ZCSIG                      0x01U
#define ZERO_ZCSIG                     0x00U

/* Current state of a trigger signal */
typedef enum {
  FALLING_ZCEVENT = -1,
  NO_ZCEVENT = 0,
  RISING_ZCEVENT = 1
} ZCEventType;

#endif                                 /* __SIMSTRUC_TYPES_H__ */
#endif                                 /* __RTWTYPES_H__ */

#ifndef MIN
#define MIN(a,b)                       ((a) < (b) ? (a) : (b))
#endif

#ifndef MAX
#define MAX(a,b)                       ((a) > (b) ? (a) : (b))
#endif
```

#### LambdaAdp.c
```c
/********************************************************************
 * COPYRIGHT -- Bernecker + Rainer Industrie-Elektronik Ges.m.b.H.
 ********************************************************************
 * Program: LambdaAdp
 * File: LambdaAdp.c
 * Author: 105051472
 * Created: Wed Oct 29 12:06:16 2014
 ********************************************************************
 * Implementation of program LambdaAdp
 ********************************************************************
 * Generated with B&R Automation Studio Target for Simulink V4.2
 * (ERT based)
 ********************************************************************/
#include "LambdaAdp.h"
#include "LambdaAdp_private.h"

/*  Defines */

/* Named constants for Chart: '<S1>/Lambda_Active' */
#define LambdaAdp_IN_Lambda_Corr_OFF   ((uint8_T)1U)
#define LambdaAdp_IN_Lambda_Corr_ON    ((uint8_T)2U)

/*  Data Types */

/**************************** GLOBAL DATA *************************************/
/*  Definitions */

/* Block signals (auto storage) */
struct BlockIO_LambdaAdp LambdaAdp_B;

/* Block states (auto storage) */
struct D_Work_LambdaAdp LambdaAdp_DWork;

/*  Declarations  */

/***************************** FILE SCOPE DATA ********************************/

/*************************** FUNCTIONS ****************************************/

/* Model step function */
void LambdaAdp_step(struct lLamCorr* inst)
{
  real32_T rtb_Divide;
  real32_T rtb_Yk1;

  /* S-Function (bur_in): '<Root>/Input4' */
  LambdaAdp_B.Input4 = inst->bLambda_Corr_Enable;

  /* S-Function (bur_in): '<Root>/Input1' */
  LambdaAdp_B.Input1 = inst->rP_Rot;

  /* S-Function (bur_in): '<Root>/Input2' */
  LambdaAdp_B.Input2 = inst->rN_Eng;

  /* S-Function (bur_in): '<Root>/Input3' */
  LambdaAdp_B.Input3 = inst->rLam_OffsLimit_Neg;

  /* Outputs for Atomic SubSystem: '<Root>/LambdaAdaption' */
  /* Product: '<S1>/Divide' incorporates:
   *  Constant: '<S1>/inst->rP_Nom'
   */
  rtb_Divide = LambdaAdp_B.Input1 / inst->rP_Nom;

  /* Product: '<S1>/Divide1' incorporates:
   *  Constant: '<S1>/inst->rN_Set'
   *  Sum: '<S1>/Subtract'
   */
  rtb_Yk1 = (LambdaAdp_B.Input2 - inst->rN_Set) / inst->rN_Set;

  /* RelationalOperator: '<S1>/Relational Operator2' incorporates:
   *  Constant: '<S1>/no_limit1'
   */
  LambdaAdp_B.RelationalOperator2 = (rtb_Yk1 <= 0.0F);

  /* RelationalOperator: '<S1>/Relational Operator' incorporates:
   *  Constant: '<S1>/inst->rP_Rot_Norm_Lam_Trig'
   */
  LambdaAdp_B.RelationalOperator = (rtb_Divide >= inst->rP_Rot_Norm_Lam_Trig);

  /* RelationalOperator: '<S1>/Relational Operator1' incorporates:
   *  Constant: '<S1>/inst->rN_Delta_Lim'
   */
  LambdaAdp_B.RelationalOperator1 = (rtb_Yk1 <= inst->rN_Delta_Lim);

  /* Chart: '<S1>/Lambda_Active' */
  /* Gateway: LambdaAdaption/Lambda_Active */
  /* During: LambdaAdaption/Lambda_Active */
  if (LambdaAdp_DWork.is_active_c1_LambdaAdp == 0U) {
    /* Entry: LambdaAdaption/Lambda_Active */
    LambdaAdp_DWork.is_active_c1_LambdaAdp = 1U;

    /* Entry Internal: LambdaAdaption/Lambda_Active */
    /* Transition: '<S2>:3' */
    LambdaAdp_DWork.is_c1_LambdaAdp = LambdaAdp_IN_Lambda_Corr_OFF;

    /* Entry 'Lambda_Corr_OFF': '<S2>:2' */
    LambdaAdp_B.bLambda_Corr_Act = FALSE;
  } else if (LambdaAdp_DWork.is_c1_LambdaAdp == LambdaAdp_IN_Lambda_Corr_OFF) {
    /* During 'Lambda_Corr_OFF': '<S2>:2' */
    if (LambdaAdp_B.RelationalOperator && LambdaAdp_B.RelationalOperator2 &&
        LambdaAdp_B.Input4) {
      /* Transition: '<S2>:4' */
      LambdaAdp_DWork.is_c1_LambdaAdp = LambdaAdp_IN_Lambda_Corr_ON;

      /* Entry 'Lambda_Corr_ON': '<S2>:6' */
      LambdaAdp_B.bLambda_Corr_Act = TRUE;
    }
  } else {
    /* During 'Lambda_Corr_ON': '<S2>:6' */
    if ((!LambdaAdp_B.RelationalOperator1) && (!LambdaAdp_B.RelationalOperator))
    {
      /* Transition: '<S2>:5' */
      LambdaAdp_DWork.is_c1_LambdaAdp = LambdaAdp_IN_Lambda_Corr_OFF;

      /* Entry 'Lambda_Corr_OFF': '<S2>:2' */
      LambdaAdp_B.bLambda_Corr_Act = FALSE;
    }
  }

  /* End of Chart: '<S1>/Lambda_Active' */

  /* Outputs for Enabled SubSystem: '<S1>/MAX' incorporates:
   *  EnablePort: '<S3>/Enable'
   */
  if (LambdaAdp_B.bLambda_Corr_Act) {
    if (!LambdaAdp_DWork.MAX_MODE) {
      /* InitializeConditions for UnitDelay: '<S3>/Unit Delay' */
      LambdaAdp_DWork.UnitDelay_DSTATE = 0.0F;
      LambdaAdp_DWork.MAX_MODE = TRUE;
    }

    /* MinMax: '<S3>/MinMax' incorporates:
     *  UnitDelay: '<S3>/Unit Delay'
     */
    if (rtb_Divide >= LambdaAdp_DWork.UnitDelay_DSTATE) {
      LambdaAdp_B.MinMax = rtb_Divide;
    } else {
      LambdaAdp_B.MinMax = LambdaAdp_DWork.UnitDelay_DSTATE;
    }

    /* End of MinMax: '<S3>/MinMax' */

    /* Update for UnitDelay: '<S3>/Unit Delay' */
    LambdaAdp_DWork.UnitDelay_DSTATE = LambdaAdp_B.MinMax;
  } else {
    if (LambdaAdp_DWork.MAX_MODE) {
      /* Disable for Outport: '<S3>/Out1' */
      LambdaAdp_B.MinMax = 0.0F;
      LambdaAdp_DWork.MAX_MODE = FALSE;
    }
  }

  /* End of Outputs for SubSystem: '<S1>/MAX' */

  /* Product: '<S1>/Product' incorporates:
   *  Constant: '<S1>/inst->rP_Rot_Norm_Lambda_Gain'
   */
  rtb_Divide = LambdaAdp_B.MinMax * inst->rP_Rot_Norm_Lambda_Gain;

  /* Switch: '<S5>/Switch2' incorporates:
   *  Constant: '<S1>/inst->rLam_OffsLimit_pos'
   *  RelationalOperator: '<S5>/LowerRelop1'
   *  RelationalOperator: '<S5>/UpperRelop'
   *  Switch: '<S5>/Switch'
   */
  if (rtb_Divide > inst->rLam_OffsLimit_pos) {
    rtb_Divide = inst->rLam_OffsLimit_pos;
  } else {
    if (rtb_Divide < LambdaAdp_B.Input3) {
      /* Switch: '<S5>/Switch' */
      rtb_Divide = LambdaAdp_B.Input3;
    }
  }

  /* End of Switch: '<S5>/Switch2' */

  /* Sum: '<S4>/Difference Inputs1' incorporates:
   *  UnitDelay: '<S4>/Delay Input2'
   */
  rtb_Yk1 = rtb_Divide - LambdaAdp_DWork.DelayInput2_DSTATE;

  /* Product: '<S4>/delta rise limit' incorporates:
   *  Constant: '<S1>/inst->rLam_Ramp_Grad'
   *  SampleTimeMath: '<S4>/sample time'
   *
   * About '<S4>/sample time':
   *  y = K where K = ( w * Ts )
   */
  rtb_Divide = inst->rLam_Ramp_Grad * 0.01F;

  /* Switch: '<S6>/Switch2' incorporates:
   *  RelationalOperator: '<S6>/LowerRelop1'
   */
  if (!(rtb_Yk1 > rtb_Divide)) {
    /* Product: '<S4>/delta fall limit' incorporates:
     *  Constant: '<S1>/no_limit'
     *  SampleTimeMath: '<S4>/sample time'
     *
     * About '<S4>/sample time':
     *  y = K where K = ( w * Ts )
     */
    rtb_Divide = -999.99F;

    /* Switch: '<S6>/Switch' incorporates:
     *  RelationalOperator: '<S6>/UpperRelop'
     */
    if (!(rtb_Yk1 < -999.99F)) {
      rtb_Divide = rtb_Yk1;
    }

    /* End of Switch: '<S6>/Switch' */
  }

  /* End of Switch: '<S6>/Switch2' */

  /* Sum: '<S4>/Difference Inputs2' incorporates:
   *  UnitDelay: '<S4>/Delay Input2'
   */
  LambdaAdp_B.DifferenceInputs2 = rtb_Divide +
    LambdaAdp_DWork.DelayInput2_DSTATE;

  /* Update for UnitDelay: '<S4>/Delay Input2' */
  LambdaAdp_DWork.DelayInput2_DSTATE = LambdaAdp_B.DifferenceInputs2;

  /* End of Outputs for SubSystem: '<Root>/LambdaAdaption' */

  /* S-Function (bur_out): '<Root>/Output' */
  inst->rLambda_Corr = LambdaAdp_B.DifferenceInputs2;

  /* S-Function (bur_out): '<Root>/Output1' */
  inst->bLambda_Freeze = LambdaAdp_B.bLambda_Corr_Act;

  /* S-Function (bur_out): '<Root>/Output2' */
  inst->rP_Rot_Max = LambdaAdp_B.MinMax;

  /* S-Function (bur_out): '<Root>/Output3' */
  inst->bN_Delta_Act = LambdaAdp_B.RelationalOperator1;

  /* S-Function (bur_out): '<Root>/Output4' */
  inst->bP_Rot_Lambda_Act = LambdaAdp_B.RelationalOperator;

  /* S-Function (bur_out): '<Root>/Output5' */
  inst->bN_Delta_Neg = LambdaAdp_B.RelationalOperator2;
}

/* Model initialize function */
void LambdaAdp_initialize(struct lLamCorr* inst)
{
  /* InitializeConditions for Atomic SubSystem: '<Root>/LambdaAdaption' */
  /* InitializeConditions for Chart: '<S1>/Lambda_Active' */
  LambdaAdp_B.bLambda_Corr_Act = FALSE;

  /* End of InitializeConditions for SubSystem: '<Root>/LambdaAdaption' */
}

/* Model terminate function */
void LambdaAdp_terminate(struct lLamCorr* inst)
{
  /* (no terminate code required) */
}

/*======================== TOOL VERSION INFORMATION ==========================*
 * MATLAB 8.0 (R2012b)20-Jul-2012                                             *
 * Simulink 8.0 (R2012b)20-Jul-2012                                           *
 * Simulink Coder 8.3 (R2012b)20-Jul-2012                                     *
 * Embedded Coder 6.3 (R2012b)20-Jul-2012                                     *
 * Stateflow 8.0 (R2012b)20-Jul-2012                                          *
 *============================================================================*/

/*======================= LICENSE IN USE INFORMATION =========================*
 * matlab                                                                     *
 * matlab_coder                                                               *
 * real-time_workshop                                                         *
 * rtw_embedded_coder                                                         *
 * simulink                                                                   *
 * stateflow                                                                  *
 *============================================================================*/
```

#### main.c
```c
/********************************************************************
 * COPYRIGHT -- Bernecker + Rainer Industrie-Elektronik Ges.m.b.H.
 ********************************************************************
 * Program: LambdaAdp
 * File: main.c
 * Author: 105051472
 * Created: Wed Oct 29 12:06:16 2014
 ********************************************************************
 * Implementation of program LambdaAdp
 ********************************************************************
 * Generated with B&R Automation Studio Target for Simulink V4.2
 * (ERT based)
 ********************************************************************/
#include <bur/plctypes.h>
#include "LambdaAdp.h"
#include "rtwtypes.h"

/* Defines */
#define SS_TERMINATE 4
#define SS_OUTPUT 3
#define SS_INITIALIZE 2

/*  Data Types */

/**************************** GLOBAL DATA *************************************/
/*  Definitions */

/*  Declarations  */

/***************************** FILE SCOPE DATA ********************************/

/*************************** FUNCTIONS ****************************************/
#ifdef __cplusplus

unsigned long bur_heap_size = 6553500;

#endif

void lLamCorr(struct lLamCorr* inst)
{

  switch (inst->ssMethodType)
  {
   case SS_INITIALIZE:
    /* call model initialize function */
    LambdaAdp_initialize(inst);
    break;

   case SS_OUTPUT:
    /* call model step function */
    LambdaAdp_step(inst);

    break;

   case SS_TERMINATE:
    /* call model terminate function */
    LambdaAdp_terminate(inst);
    break;
  }
}

/*****************************************************************************
   Function block sample time: 0.01s
 *****************************************************************************/

/*****************************************************************************
   B&R Automation Studio Target for Simulink Version: A4.3.1 (09-Apr-2014)
 *****************************************************************************/

/*======================== TOOL VERSION INFORMATION ==========================*
 * MATLAB 8.0 (R2012b)20-Jul-2012                                             *
 * Simulink 8.0 (R2012b)20-Jul-2012                                           *
 * Simulink Coder 8.3 (R2012b)20-Jul-2012                                     *
 * Embedded Coder 6.3 (R2012b)20-Jul-2012                                     *
 * Stateflow 8.0 (R2012b)20-Jul-2012                                          *
 *============================================================================*/

/*======================= LICENSE IN USE INFORMATION =========================*
 * matlab                                                                     *
 * matlab_coder                                                               *
 * real-time_workshop                                                         *
 * rtw_embedded_coder                                                         *
 * simulink                                                                   *
 * stateflow                                                                  *
 *============================================================================*/
```

#### lib_properties.txt
```
For manual assignment to hardware configuration please
add the following additional include directories:

\Logical\MATLAB_includes\R2012b\

And the following additional build options:

-lm -D MODEL=LambdaAdp -D NUMST=1 -D NCSTATES=0 -D HAVESTDIO -D ONESTEPFCN=1 -D TERMFCN=1 -D MAT_FILE=0 -D MULTI_INSTANCE_CODE=0 -D INTEGER_CODE=0 -D MT=0 -D CLASSIC_INTERFACE=0 -D TID01EQ=0
```

### bio_sig.h
```c
/*
 * Copyright 1994-2002 The MathWorks, Inc.
 *
 * File: bio_sig.h     $Revision: 1.10 $
 *
 * Abstract:
 *	typedef for BlockIOSignals, included by *rt_main.c and MODEL.bio
 */

#ifndef _BIO_SIG_H_
# define _BIO_SIG_H_

typedef struct BlockIOSignals_tag {
  char_T   *blockName;    /* Block's full path name (RTW mangled version)     */
  char_T   *signalName;   /* Signal label (unmangled, or NULL if not present) */
  uint_T   portNumber;    /* Block output port number (starting at 0)         */
  uint_T   signalWidth;   /* Signal's width                                   */
  void     *signalAddr;   /* Signal's Address in the block I/O vector         */
  char_T   *dtName;       /* The C-language data type name                    */
  uint_T   dtSize;        /* The size in # of bytes for the data type         */
} BlockIOSignals;

#endif
```

### blas.h
```c
/*
 * @(#)blas.h    generated by: makeheader 5.1.5  Tue May 24 21:10:39 2011
 *
 *		built from:	../include/copyright.h
 *				//mathworks/hub/3rdparty/R2011b/280239/glnx86/REFBLAS/include/blas.h
 */

#if defined(_MSC_VER)
# pragma once
#endif
#if defined(__GNUC__) && (__GNUC__ > 3 || (__GNUC__ == 3 && __GNUC_MINOR__ > 3))
# pragma once
#endif

#ifndef blas_h
#define blas_h

/*
 * Copyright 1984-2003 The MathWorks, Inc.
 * All Rights Reserved.
 */

/*
 *  Header File include/blas.h
 *  Auto generated by f2h.pl, do not modify by hand
 */

#if defined(_WIN32) || defined(__hpux)
#define FORTRAN_WRAPPER(x) x
#else
#define FORTRAN_WRAPPER(x) x ## _
#endif

#ifndef COMPLEX_TYPES
#define COMPLEX_TYPES
  typedef struct{float r,i;} complex;
  typedef struct{double r,i;} doublecomplex;
#endif

#ifdef __cplusplus
    extern "C" {
#endif

/* Source: caxpy.f */
#define caxpy FORTRAN_WRAPPER(caxpy)
extern void caxpy(
    ptrdiff_t *n,
    float  *ca,
    float  *cx,
    ptrdiff_t *incx,
    float  *cy,
    ptrdiff_t *incy
);

/* Source: ccopy.f */
#define ccopy FORTRAN_WRAPPER(ccopy)
extern void ccopy(
    ptrdiff_t *n,
    float  *cx,
    ptrdiff_t *incx,
    float  *cy,
    ptrdiff_t *incy
);

/* Source: cdotc.f */
#define cdotc FORTRAN_WRAPPER(cdotc)
#ifndef FORTRAN_COMPLEX_FUNCTIONS_RETURN_VOID
extern complex cdotc(
#else
extern void cdotc(
    complex* retval,
#endif
    ptrdiff_t *n,
    float  *cx,
    ptrdiff_t *incx,
    float  *cy,
    ptrdiff_t *incy
);

/* Source: cdotu.f */
#define cdotu FORTRAN_WRAPPER(cdotu)
#ifndef FORTRAN_COMPLEX_FUNCTIONS_RETURN_VOID
extern complex cdotu(
#else
extern void cdotu(
    complex* retval,
#endif
    ptrdiff_t *n,
    float  *cx,
    ptrdiff_t *incx,
    float  *cy,
    ptrdiff_t *incy
);

/* Source: cgbmv.f */
#define cgbmv FORTRAN_WRAPPER(cgbmv)
extern void cgbmv(
    char   *trans,
    ptrdiff_t *m,
    ptrdiff_t *n,
    ptrdiff_t *kl,
    ptrdiff_t *ku,
    float  *alpha,
    float  *a,
    ptrdiff_t *lda,
    float  *x,
    ptrdiff_t *incx,
    float  *beta,
    float  *y,
    ptrdiff_t *incy
);

/* Source: cgemm.f */
#define cgemm FORTRAN_WRAPPER(cgemm)
extern void cgemm(
    char   *transa,
    char   *transb,
    ptrdiff_t *m,
    ptrdiff_t *n,
    ptrdiff_t *k,
    float  *alpha,
    float  *a,
    ptrdiff_t *lda,
    float  *b,
    ptrdiff_t *ldb,
    float  *beta,
    float  *c,
    ptrdiff_t *ldc
);

/* Source: cgemv.f */
#define cgemv FORTRAN_WRAPPER(cgemv)
extern void cgemv(
    char   *trans,
    ptrdiff_t *m,
    ptrdiff_t *n,
    float  *alpha,
    float  *a,
    ptrdiff_t *lda,
    float  *x,
    ptrdiff_t *incx,
    float  *beta,
    float  *y,
    ptrdiff_t *incy
);

/* Source: cgerc.f */
#define cgerc FORTRAN_WRAPPER(cgerc)
extern void cgerc(
    ptrdiff_t *m,
    ptrdiff_t *n,
    float  *alpha,
    float  *x,
    ptrdiff_t *incx,
    float  *y,
    ptrdiff_t *incy,
    float  *a,
    ptrdiff_t *lda
);

/* Source: cgeru.f */
#define cgeru FORTRAN_WRAPPER(cgeru)
extern void cgeru(
    ptrdiff_t *m,
    ptrdiff_t *n,
    float  *alpha,
    float  *x,
    ptrdiff_t *incx,
    float  *y,
    ptrdiff_t *incy,
    float  *a,
    ptrdiff_t *lda
);

/* Source: chbmv.f */
#define chbmv FORTRAN_WRAPPER(chbmv)
extern void chbmv(
    char   *uplo,
    ptrdiff_t *n,
    ptrdiff_t *k,
    float  *alpha,
    float  *a,
    ptrdiff_t *lda,
    float  *x,
    ptrdiff_t *incx,
    float  *beta,
    float  *y,
    ptrdiff_t *incy
);

/* Source: chemm.f */
#define chemm FORTRAN_WRAPPER(chemm)
extern void chemm(
    char   *side,
    char   *uplo,
    ptrdiff_t *m,
    ptrdiff_t *n,
    float  *alpha,
    float  *a,
    ptrdiff_t *lda,
    float  *b,
    ptrdiff_t *ldb,
    float  *beta,
    float  *c,
    ptrdiff_t *ldc
);

/* Source: chemv.f */
#define chemv FORTRAN_WRAPPER(chemv)
extern void chemv(
    char   *uplo,
    ptrdiff_t *n,
    float  *alpha,
    float  *a,
    ptrdiff_t *lda,
    float  *x,
    ptrdiff_t *incx,
    float  *beta,
    float  *y,
    ptrdiff_t *incy
);

/* Source: cher.f */
#define cher FORTRAN_WRAPPER(cher)
extern void cher(
    char   *uplo,
    ptrdiff_t *n,
    float  *alpha,
    float  *x,
    ptrdiff_t *incx,
    float  *a,
    ptrdiff_t *lda
);

/* Source: cher2.f */
#define cher2 FORTRAN_WRAPPER(cher2)
extern void cher2(
    char   *uplo,
    ptrdiff_t *n,
    float  *alpha,
    float  *x,
    ptrdiff_t *incx,
    float  *y,
    ptrdiff_t *incy,
    float  *a,
    ptrdiff_t *lda
);

/* Source: cher2k.f */
#define cher2k FORTRAN_WRAPPER(cher2k)
extern void cher2k(
    char   *uplo,
    char   *trans,
    ptrdiff_t *n,
    ptrdiff_t *k,
    float  *alpha,
    float  *a,
    ptrdiff_t *lda,
    float  *b,
    ptrdiff_t *ldb,
    float  *beta,
    float  *c,
    ptrdiff_t *ldc
);

/* Source: cherk.f */
#define cherk FORTRAN_WRAPPER(cherk)
extern void cherk(
    char   *uplo,
    char   *trans,
    ptrdiff_t *n,
    ptrdiff_t *k,
    float  *alpha,
    float  *a,
    ptrdiff_t *lda,
    float  *beta,
    float  *c,
    ptrdiff_t *ldc
);

/* Source: chpmv.f */
#define chpmv FORTRAN_WRAPPER(chpmv)
extern void chpmv(
    char   *uplo,
    ptrdiff_t *n,
    float  *alpha,
    float  *ap,
    float  *x,
    ptrdiff_t *incx,
    float  *beta,
    float  *y,
    ptrdiff_t *incy
);

/* Source: chpr.f */
#define chpr FORTRAN_WRAPPER(chpr)
extern void chpr(
    char   *uplo,
    ptrdiff_t *n,
    float  *alpha,
    float  *x,
    ptrdiff_t *incx,
    float  *ap
);

/* Source: chpr2.f */
#define chpr2 FORTRAN_WRAPPER(chpr2)
extern void chpr2(
    char   *uplo,
    ptrdiff_t *n,
    float  *alpha,
    float  *x,
    ptrdiff_t *incx,
    float  *y,
    ptrdiff_t *incy,
    float  *ap
);

/* Source: crotg.f */
#define crotg FORTRAN_WRAPPER(crotg)
extern void crotg(
    float  *ca,
    float  *cb,
    float  *c,
    float  *s
);

/* Source: cscal.f */
#define cscal FORTRAN_WRAPPER(cscal)
extern void cscal(
    ptrdiff_t *n,
    float  *ca,
    float  *cx,
    ptrdiff_t *incx
);

/* Source: csrot.f */
#define csrot FORTRAN_WRAPPER(csrot)
extern void csrot(
    ptrdiff_t *n,
    float  *cx,
    ptrdiff_t *incx,
    float  *cy,
    ptrdiff_t *incy,
    float  *c,
    float  *s
);

/* Source: csscal.f */
#define csscal FORTRAN_WRAPPER(csscal)
extern void csscal(
    ptrdiff_t *n,
    float  *sa,
    float  *cx,
    ptrdiff_t *incx
);

/* Source: cswap.f */
#define cswap FORTRAN_WRAPPER(cswap)
extern void cswap(
    ptrdiff_t *n,
    float  *cx,
    ptrdiff_t *incx,
    float  *cy,
    ptrdiff_t *incy
);

/* Source: csymm.f */
#define csymm FORTRAN_WRAPPER(csymm)
extern void csymm(
    char   *side,
    char   *uplo,
    ptrdiff_t *m,
    ptrdiff_t *n,
    float  *alpha,
    float  *a,
    ptrdiff_t *lda,
    float  *b,
    ptrdiff_t *ldb,
    float  *beta,
    float  *c,
    ptrdiff_t *ldc
);

/* Source: csyr2k.f */
#define csyr2k FORTRAN_WRAPPER(csyr2k)
extern void csyr2k(
    char   *uplo,
    char   *trans,
    ptrdiff_t *n,
    ptrdiff_t *k,
    float  *alpha,
    float  *a,
    ptrdiff_t *lda,
    float  *b,
    ptrdiff_t *ldb,
    float  *beta,
    float  *c,
    ptrdiff_t *ldc
);

/* Source: csyrk.f */
#define csyrk FORTRAN_WRAPPER(csyrk)
extern void csyrk(
    char   *uplo,
    char   *trans,
    ptrdiff_t *n,
    ptrdiff_t *k,
    float  *alpha,
    float  *a,
    ptrdiff_t *lda,
    float  *beta,
    float  *c,
    ptrdiff_t *ldc
);

/* Source: ctbmv.f */
#define ctbmv FORTRAN_WRAPPER(ctbmv)
extern void ctbmv(
    char   *uplo,
    char   *trans,
    char   *diag,
    ptrdiff_t *n,
    ptrdiff_t *k,
    float  *a,
    ptrdiff_t *lda,
    float  *x,
    ptrdiff_t *incx
);

/* Source: ctbsv.f */
#define ctbsv FORTRAN_WRAPPER(ctbsv)
extern void ctbsv(
    char   *uplo,
    char   *trans,
    char   *diag,
    ptrdiff_t *n,
    ptrdiff_t *k,
    float  *a,
    ptrdiff_t *lda,
    float  *x,
    ptrdiff_t *incx
);

/* Source: ctpmv.f */
#define ctpmv FORTRAN_WRAPPER(ctpmv)
extern void ctpmv(
    char   *uplo,
    char   *trans,
    char   *diag,
    ptrdiff_t *n,
    float  *ap,
    float  *x,
    ptrdiff_t *incx
);

/* Source: ctpsv.f */
#define ctpsv FORTRAN_WRAPPER(ctpsv)
extern void ctpsv(
    char   *uplo,
    char   *trans,
    char   *diag,
    ptrdiff_t *n,
    float  *ap,
    float  *x,
    ptrdiff_t *incx
);

/* Source: ctrmm.f */
#define ctrmm FORTRAN_WRAPPER(ctrmm)
extern void ctrmm(
    char   *side,
    char   *uplo,
    char   *transa,
    char   *diag,
    ptrdiff_t *m,
    ptrdiff_t *n,
    float  *alpha,
    float  *a,
    ptrdiff_t *lda,
    float  *b,
    ptrdiff_t *ldb
);

/* Source: ctrmv.f */
#define ctrmv FORTRAN_WRAPPER(ctrmv)
extern void ctrmv(
    char   *uplo,
    char   *trans,
    char   *diag,
    ptrdiff_t *n,
    float  *a,
    ptrdiff_t *lda,
    float  *x,
    ptrdiff_t *incx
);

/* Source: ctrsm.f */
#define ctrsm FORTRAN_WRAPPER(ctrsm)
extern void ctrsm(
    char   *side,
    char   *uplo,
    char   *transa,
    char   *diag,
    ptrdiff_t *m,
    ptrdiff_t *n,
    float  *alpha,
    float  *a,
    ptrdiff_t *lda,
    float  *b,
    ptrdiff_t *ldb
);

/* Source: ctrsv.f */
#define ctrsv FORTRAN_WRAPPER(ctrsv)
extern void ctrsv(
    char   *uplo,
    char   *trans,
    char   *diag,
    ptrdiff_t *n,
    float  *a,
    ptrdiff_t *lda,
    float  *x,
    ptrdiff_t *incx
);

/* Source: dasum.f */
#define dasum FORTRAN_WRAPPER(dasum)
extern double dasum(
    ptrdiff_t *n,
    double *dx,
    ptrdiff_t *incx
);

/* Source: daxpy.f */
#define daxpy FORTRAN_WRAPPER(daxpy)
extern void daxpy(
    ptrdiff_t *n,
    double *da,
    double *dx,
    ptrdiff_t *incx,
    double *dy,
    ptrdiff_t *incy
);

/* Source: dcabs1.f */
#define dcabs1 FORTRAN_WRAPPER(dcabs1)
extern double dcabs1(
    double *z
);

/* Source: dcopy.f */
#define dcopy FORTRAN_WRAPPER(dcopy)
extern void dcopy(
    ptrdiff_t *n,
    double *dx,
    ptrdiff_t *incx,
    double *dy,
    ptrdiff_t *incy
);

/* Source: ddot.f */
#define ddot FORTRAN_WRAPPER(ddot)
extern double ddot(
    ptrdiff_t *n,
    double *dx,
    ptrdiff_t *incx,
    double *dy,
    ptrdiff_t *incy
);

/* Source: dgbmv.f */
#define dgbmv FORTRAN_WRAPPER(dgbmv)
extern void dgbmv(
    char   *trans,
    ptrdiff_t *m,
    ptrdiff_t *n,
    ptrdiff_t *kl,
    ptrdiff_t *ku,
    double *alpha,
    double *a,
    ptrdiff_t *lda,
    double *x,
    ptrdiff_t *incx,
    double *beta,
    double *y,
    ptrdiff_t *incy
);

/* Source: dgemm.f */
#define dgemm FORTRAN_WRAPPER(dgemm)
extern void dgemm(
    char   *transa,
    char   *transb,
    ptrdiff_t *m,
    ptrdiff_t *n,
    ptrdiff_t *k,
    double *alpha,
    double *a,
    ptrdiff_t *lda,
    double *b,
    ptrdiff_t *ldb,
    double *beta,
    double *c,
    ptrdiff_t *ldc
);

/* Source: dgemv.f */
#define dgemv FORTRAN_WRAPPER(dgemv)
extern void dgemv(
    char   *trans,
    ptrdiff_t *m,
    ptrdiff_t *n,
    double *alpha,
    double *a,
    ptrdiff_t *lda,
    double *x,
    ptrdiff_t *incx,
    double *beta,
    double *y,
    ptrdiff_t *incy
);

/* Source: dger.f */
#define dger FORTRAN_WRAPPER(dger)
extern void dger(
    ptrdiff_t *m,
    ptrdiff_t *n,
    double *alpha,
    double *x,
    ptrdiff_t *incx,
    double *y,
    ptrdiff_t *incy,
    double *a,
    ptrdiff_t *lda
);

/* Source: dnrm2.f */
#define dnrm2 FORTRAN_WRAPPER(dnrm2)
extern double dnrm2(
    ptrdiff_t *n,
    double *x,
    ptrdiff_t *incx
);

/* Source: drot.f */
#define drot FORTRAN_WRAPPER(drot)
extern void drot(
    ptrdiff_t *n,
    double *dx,
    ptrdiff_t *incx,
    double *dy,
    ptrdiff_t *incy,
    double *c,
    double *s
);

/* Source: drotg.f */
#define drotg FORTRAN_WRAPPER(drotg)
extern void drotg(
    double *da,
    double *db,
    double *c,
    double *s
);

/* Source: drotm.f */
#define drotm FORTRAN_WRAPPER(drotm)
extern void drotm(
    ptrdiff_t *n,
    double *dx,
    ptrdiff_t *incx,
    double *dy,
    ptrdiff_t *incy,
    double *dparam
);

/* Source: drotmg.f */
#define drotmg FORTRAN_WRAPPER(drotmg)
extern void drotmg(
    double *dd1,
    double *dd2,
    double *dx1,
    double *dy1,
    double *dparam
);

/* Source: dsbmv.f */
#define dsbmv FORTRAN_WRAPPER(dsbmv)
extern void dsbmv(
    char   *uplo,
    ptrdiff_t *n,
    ptrdiff_t *k,
    double *alpha,
    double *a,
    ptrdiff_t *lda,
    double *x,
    ptrdiff_t *incx,
    double *beta,
    double *y,
    ptrdiff_t *incy
);

/* Source: dscal.f */
#define dscal FORTRAN_WRAPPER(dscal)
extern void dscal(
    ptrdiff_t *n,
    double *da,
    double *dx,
    ptrdiff_t *incx
);

/* Source: dsdot.f */
#define dsdot FORTRAN_WRAPPER(dsdot)
extern double dsdot(
    ptrdiff_t *n,
    float  *sx,
    ptrdiff_t *incx,
    float  *sy,
    ptrdiff_t *incy
);

/* Source: dspmv.f */
#define dspmv FORTRAN_WRAPPER(dspmv)
extern void dspmv(
    char   *uplo,
    ptrdiff_t *n,
    double *alpha,
    double *ap,
    double *x,
    ptrdiff_t *incx,
    double *beta,
    double *y,
    ptrdiff_t *incy
);

/* Source: dspr.f */
#define dspr FORTRAN_WRAPPER(dspr)
extern void dspr(
    char   *uplo,
    ptrdiff_t *n,
    double *alpha,
    double *x,
    ptrdiff_t *incx,
    double *ap
);

/* Source: dspr2.f */
#define dspr2 FORTRAN_WRAPPER(dspr2)
extern void dspr2(
    char   *uplo,
    ptrdiff_t *n,
    double *alpha,
    double *x,
    ptrdiff_t *incx,
    double *y,
    ptrdiff_t *incy,
    double *ap
);

/* Source: dswap.f */
#define dswap FORTRAN_WRAPPER(dswap)
extern void dswap(
    ptrdiff_t *n,
    double *dx,
    ptrdiff_t *incx,
    double *dy,
    ptrdiff_t *incy
);

/* Source: dsymm.f */
#define dsymm FORTRAN_WRAPPER(dsymm)
extern void dsymm(
    char   *side,
    char   *uplo,
    ptrdiff_t *m,
    ptrdiff_t *n,
    double *alpha,
    double *a,
    ptrdiff_t *lda,
    double *b,
    ptrdiff_t *ldb,
    double *beta,
    double *c,
    ptrdiff_t *ldc
);

/* Source: dsymv.f */
#define dsymv FORTRAN_WRAPPER(dsymv)
extern void dsymv(
    char   *uplo,
    ptrdiff_t *n,
    double *alpha,
    double *a,
    ptrdiff_t *lda,
    double *x,
    ptrdiff_t *incx,
    double *beta,
    double *y,
    ptrdiff_t *incy
);

/* Source: dsyr.f */
#define dsyr FORTRAN_WRAPPER(dsyr)
extern void dsyr(
    char   *uplo,
    ptrdiff_t *n,
    double *alpha,
    double *x,
    ptrdiff_t *incx,
    double *a,
    ptrdiff_t *lda
);

/* Source: dsyr2.f */
#define dsyr2 FORTRAN_WRAPPER(dsyr2)
extern void dsyr2(
    char   *uplo,
    ptrdiff_t *n,
    double *alpha,
    double *x,
    ptrdiff_t *incx,
    double *y,
    ptrdiff_t *incy,
    double *a,
    ptrdiff_t *lda
);

/* Source: dsyr2k.f */
#define dsyr2k FORTRAN_WRAPPER(dsyr2k)
extern void dsyr2k(
    char   *uplo,
    char   *trans,
    ptrdiff_t *n,
    ptrdiff_t *k,
    double *alpha,
    double *a,
    ptrdiff_t *lda,
    double *b,
    ptrdiff_t *ldb,
    double *beta,
    double *c,
    ptrdiff_t *ldc
);

/* Source: dsyrk.f */
#define dsyrk FORTRAN_WRAPPER(dsyrk)
extern void dsyrk(
    char   *uplo,
    char   *trans,
    ptrdiff_t *n,
    ptrdiff_t *k,
    double *alpha,
    double *a,
    ptrdiff_t *lda,
    double *beta,
    double *c,
    ptrdiff_t *ldc
);

/* Source: dtbmv.f */
#define dtbmv FORTRAN_WRAPPER(dtbmv)
extern void dtbmv(
    char   *uplo,
    char   *trans,
    char   *diag,
    ptrdiff_t *n,
    ptrdiff_t *k,
    double *a,
    ptrdiff_t *lda,
    double *x,
    ptrdiff_t *incx
);

/* Source: dtbsv.f */
#define dtbsv FORTRAN_WRAPPER(dtbsv)
extern void dtbsv(
    char   *uplo,
    char   *trans,
    char   *diag,
    ptrdiff_t *n,
    ptrdiff_t *k,
    double *a,
    ptrdiff_t *lda,
    double *x,
    ptrdiff_t *incx
);

/* Source: dtpmv.f */
#define dtpmv FORTRAN_WRAPPER(dtpmv)
extern void dtpmv(
    char   *uplo,
    char   *trans,
    char   *diag,
    ptrdiff_t *n,
    double *ap,
    double *x,
    ptrdiff_t *incx
);

/* Source: dtpsv.f */
#define dtpsv FORTRAN_WRAPPER(dtpsv)
extern void dtpsv(
    char   *uplo,
    char   *trans,
    char   *diag,
    ptrdiff_t *n,
    double *ap,
    double *x,
    ptrdiff_t *incx
);

/* Source: dtrmm.f */
#define dtrmm FORTRAN_WRAPPER(dtrmm)
extern void dtrmm(
    char   *side,
    char   *uplo,
    char   *transa,
    char   *diag,
    ptrdiff_t *m,
    ptrdiff_t *n,
    double *alpha,
    double *a,
    ptrdiff_t *lda,
    double *b,
    ptrdiff_t *ldb
);

/* Source: dtrmv.f */
#define dtrmv FORTRAN_WRAPPER(dtrmv)
extern void dtrmv(
    char   *uplo,
    char   *trans,
    char   *diag,
    ptrdiff_t *n,
    double *a,
    ptrdiff_t *lda,
    double *x,
    ptrdiff_t *incx
);

/* Source: dtrsm.f */
#define dtrsm FORTRAN_WRAPPER(dtrsm)
extern void dtrsm(
    char   *side,
    char   *uplo,
    char   *transa,
    char   *diag,
    ptrdiff_t *m,
    ptrdiff_t *n,
    double *alpha,
    double *a,
    ptrdiff_t *lda,
    double *b,
    ptrdiff_t *ldb
);

/* Source: dtrsv.f */
#define dtrsv FORTRAN_WRAPPER(dtrsv)
extern void dtrsv(
    char   *uplo,
    char   *trans,
    char   *diag,
    ptrdiff_t *n,
    double *a,
    ptrdiff_t *lda,
    double *x,
    ptrdiff_t *incx
);

/* Source: dzasum.f */
#define dzasum FORTRAN_WRAPPER(dzasum)
extern double dzasum(
    ptrdiff_t *n,
    double *zx,
    ptrdiff_t *incx
);

/* Source: dznrm2.f */
#define dznrm2 FORTRAN_WRAPPER(dznrm2)
extern double dznrm2(
    ptrdiff_t *n,
    double *x,
    ptrdiff_t *incx
);

/* Source: icamax.f */
#define icamax FORTRAN_WRAPPER(icamax)
extern ptrdiff_t icamax(
    ptrdiff_t *n,
    float  *cx,
    ptrdiff_t *incx
);

/* Source: idamax.f */
#define idamax FORTRAN_WRAPPER(idamax)
extern ptrdiff_t idamax(
    ptrdiff_t *n,
    double *dx,
    ptrdiff_t *incx
);

/* Source: isamax.f */
#define isamax FORTRAN_WRAPPER(isamax)
extern ptrdiff_t isamax(
    ptrdiff_t *n,
    float  *sx,
    ptrdiff_t *incx
);

/* Source: izamax.f */
#define izamax FORTRAN_WRAPPER(izamax)
extern ptrdiff_t izamax(
    ptrdiff_t *n,
    double *zx,
    ptrdiff_t *incx
);

/* Source: lsame.f */
#define lsame FORTRAN_WRAPPER(lsame)
extern ptrdiff_t lsame(
    char   *ca,
    char   *cb
);

/* Source: sasum.f */
#define sasum FORTRAN_WRAPPER(sasum)
#ifdef FORTRAN_FLOAT_FUNCTIONS_RETURN_DOUBLE
extern double sasum(
#else
extern float sasum(
#endif
    ptrdiff_t *n,
    float  *sx,
    ptrdiff_t *incx
);

/* Source: saxpy.f */
#define saxpy FORTRAN_WRAPPER(saxpy)
extern void saxpy(
    ptrdiff_t *n,
    float  *sa,
    float  *sx,
    ptrdiff_t *incx,
    float  *sy,
    ptrdiff_t *incy
);

/* Source: scasum.f */
#define scasum FORTRAN_WRAPPER(scasum)
#ifdef FORTRAN_FLOAT_FUNCTIONS_RETURN_DOUBLE
extern double scasum(
#else
extern float scasum(
#endif
    ptrdiff_t *n,
    float  *cx,
    ptrdiff_t *incx
);

/* Source: scnrm2.f */
#define scnrm2 FORTRAN_WRAPPER(scnrm2)
#ifdef FORTRAN_FLOAT_FUNCTIONS_RETURN_DOUBLE
extern double scnrm2(
#else
extern float scnrm2(
#endif
    ptrdiff_t *n,
    float  *x,
    ptrdiff_t *incx
);

/* Source: scopy.f */
#define scopy FORTRAN_WRAPPER(scopy)
extern void scopy(
    ptrdiff_t *n,
    float  *sx,
    ptrdiff_t *incx,
    float  *sy,
    ptrdiff_t *incy
);

/* Source: sdot.f */
#define sdot FORTRAN_WRAPPER(sdot)
#ifdef FORTRAN_FLOAT_FUNCTIONS_RETURN_DOUBLE
extern double sdot(
#else
extern float sdot(
#endif
    ptrdiff_t *n,
    float  *sx,
    ptrdiff_t *incx,
    float  *sy,
    ptrdiff_t *incy
);

/* Source: sdsdot.f */
#define sdsdot FORTRAN_WRAPPER(sdsdot)
#ifdef FORTRAN_FLOAT_FUNCTIONS_RETURN_DOUBLE
extern double sdsdot(
#else
extern float sdsdot(
#endif
    ptrdiff_t *n,
    float  *sb,
    float  *sx,
    ptrdiff_t *incx,
    float  *sy,
    ptrdiff_t *incy
);

/* Source: sgbmv.f */
#define sgbmv FORTRAN_WRAPPER(sgbmv)
extern void sgbmv(
    char   *trans,
    ptrdiff_t *m,
    ptrdiff_t *n,
    ptrdiff_t *kl,
    ptrdiff_t *ku,
    float  *alpha,
    float  *a,
    ptrdiff_t *lda,
    float  *x,
    ptrdiff_t *incx,
    float  *beta,
    float  *y,
    ptrdiff_t *incy
);

/* Source: sgemm.f */
#define sgemm FORTRAN_WRAPPER(sgemm)
extern void sgemm(
    char   *transa,
    char   *transb,
    ptrdiff_t *m,
    ptrdiff_t *n,
    ptrdiff_t *k,
    float  *alpha,
    float  *a,
    ptrdiff_t *lda,
    float  *b,
    ptrdiff_t *ldb,
    float  *beta,
    float  *c,
    ptrdiff_t *ldc
);

/* Source: sgemv.f */
#define sgemv FORTRAN_WRAPPER(sgemv)
extern void sgemv(
    char   *trans,
    ptrdiff_t *m,
    ptrdiff_t *n,
    float  *alpha,
    float  *a,
    ptrdiff_t *lda,
    float  *x,
    ptrdiff_t *incx,
    float  *beta,
    float  *y,
    ptrdiff_t *incy
);

/* Source: sger.f */
#define sger FORTRAN_WRAPPER(sger)
extern void sger(
    ptrdiff_t *m,
    ptrdiff_t *n,
    float  *alpha,
    float  *x,
    ptrdiff_t *incx,
    float  *y,
    ptrdiff_t *incy,
    float  *a,
    ptrdiff_t *lda
);

/* Source: snrm2.f */
#define snrm2 FORTRAN_WRAPPER(snrm2)
#ifdef FORTRAN_FLOAT_FUNCTIONS_RETURN_DOUBLE
extern double snrm2(
#else
extern float snrm2(
#endif
    ptrdiff_t *n,
    float  *x,
    ptrdiff_t *incx
);

/* Source: srot.f */
#define srot FORTRAN_WRAPPER(srot)
extern void srot(
    ptrdiff_t *n,
    float  *sx,
    ptrdiff_t *incx,
    float  *sy,
    ptrdiff_t *incy,
    float  *c,
    float  *s
);

/* Source: srotg.f */
#define srotg FORTRAN_WRAPPER(srotg)
extern void srotg(
    float  *sa,
    float  *sb,
    float  *c,
    float  *s
);

/* Source: srotm.f */
#define srotm FORTRAN_WRAPPER(srotm)
extern void srotm(
    ptrdiff_t *n,
    float  *sx,
    ptrdiff_t *incx,
    float  *sy,
    ptrdiff_t *incy,
    float  *sparam
);

/* Source: srotmg.f */
#define srotmg FORTRAN_WRAPPER(srotmg)
extern void srotmg(
    float  *sd1,
    float  *sd2,
    float  *sx1,
    float  *sy1,
    float  *sparam
);

/* Source: ssbmv.f */
#define ssbmv FORTRAN_WRAPPER(ssbmv)
extern void ssbmv(
    char   *uplo,
    ptrdiff_t *n,
    ptrdiff_t *k,
    float  *alpha,
    float  *a,
    ptrdiff_t *lda,
    float  *x,
    ptrdiff_t *incx,
    float  *beta,
    float  *y,
    ptrdiff_t *incy
);

/* Source: sscal.f */
#define sscal FORTRAN_WRAPPER(sscal)
extern void sscal(
    ptrdiff_t *n,
    float  *sa,
    float  *sx,
    ptrdiff_t *incx
);

/* Source: sspmv.f */
#define sspmv FORTRAN_WRAPPER(sspmv)
extern void sspmv(
    char   *uplo,
    ptrdiff_t *n,
    float  *alpha,
    float  *ap,
    float  *x,
    ptrdiff_t *incx,
    float  *beta,
    float  *y,
    ptrdiff_t *incy
);

/* Source: sspr.f */
#define sspr FORTRAN_WRAPPER(sspr)
extern void sspr(
    char   *uplo,
    ptrdiff_t *n,
    float  *alpha,
    float  *x,
    ptrdiff_t *incx,
    float  *ap
);

/* Source: sspr2.f */
#define sspr2 FORTRAN_WRAPPER(sspr2)
extern void sspr2(
    char   *uplo,
    ptrdiff_t *n,
    float  *alpha,
    float  *x,
    ptrdiff_t *incx,
    float  *y,
    ptrdiff_t *incy,
    float  *ap
);

/* Source: sswap.f */
#define sswap FORTRAN_WRAPPER(sswap)
extern void sswap(
    ptrdiff_t *n,
    float  *sx,
    ptrdiff_t *incx,
    float  *sy,
    ptrdiff_t *incy
);

/* Source: ssymm.f */
#define ssymm FORTRAN_WRAPPER(ssymm)
extern void ssymm(
    char   *side,
    char   *uplo,
    ptrdiff_t *m,
    ptrdiff_t *n,
    float  *alpha,
    float  *a,
    ptrdiff_t *lda,
    float  *b,
    ptrdiff_t *ldb,
    float  *beta,
    float  *c,
    ptrdiff_t *ldc
);

/* Source: ssymv.f */
#define ssymv FORTRAN_WRAPPER(ssymv)
extern void ssymv(
    char   *uplo,
    ptrdiff_t *n,
    float  *alpha,
    float  *a,
    ptrdiff_t *lda,
    float  *x,
    ptrdiff_t *incx,
    float  *beta,
    float  *y,
    ptrdiff_t *incy
);

/* Source: ssyr.f */
#define ssyr FORTRAN_WRAPPER(ssyr)
extern void ssyr(
    char   *uplo,
    ptrdiff_t *n,
    float  *alpha,
    float  *x,
    ptrdiff_t *incx,
    float  *a,
    ptrdiff_t *lda
);

/* Source: ssyr2.f */
#define ssyr2 FORTRAN_WRAPPER(ssyr2)
extern void ssyr2(
    char   *uplo,
    ptrdiff_t *n,
    float  *alpha,
    float  *x,
    ptrdiff_t *incx,
    float  *y,
    ptrdiff_t *incy,
    float  *a,
    ptrdiff_t *lda
);

/* Source: ssyr2k.f */
#define ssyr2k FORTRAN_WRAPPER(ssyr2k)
extern void ssyr2k(
    char   *uplo,
    char   *trans,
    ptrdiff_t *n,
    ptrdiff_t *k,
    float  *alpha,
    float  *a,
    ptrdiff_t *lda,
    float  *b,
    ptrdiff_t *ldb,
    float  *beta,
    float  *c,
    ptrdiff_t *ldc
);

/* Source: ssyrk.f */
#define ssyrk FORTRAN_WRAPPER(ssyrk)
extern void ssyrk(
    char   *uplo,
    char   *trans,
    ptrdiff_t *n,
    ptrdiff_t *k,
    float  *alpha,
    float  *a,
    ptrdiff_t *lda,
    float  *beta,
    float  *c,
    ptrdiff_t *ldc
);

/* Source: stbmv.f */
#define stbmv FORTRAN_WRAPPER(stbmv)
extern void stbmv(
    char   *uplo,
    char   *trans,
    char   *diag,
    ptrdiff_t *n,
    ptrdiff_t *k,
    float  *a,
    ptrdiff_t *lda,
    float  *x,
    ptrdiff_t *incx
);

/* Source: stbsv.f */
#define stbsv FORTRAN_WRAPPER(stbsv)
extern void stbsv(
    char   *uplo,
    char   *trans,
    char   *diag,
    ptrdiff_t *n,
    ptrdiff_t *k,
    float  *a,
    ptrdiff_t *lda,
    float  *x,
    ptrdiff_t *incx
);

/* Source: stpmv.f */
#define stpmv FORTRAN_WRAPPER(stpmv)
extern void stpmv(
    char   *uplo,
    char   *trans,
    char   *diag,
    ptrdiff_t *n,
    float  *ap,
    float  *x,
    ptrdiff_t *incx
);

/* Source: stpsv.f */
#define stpsv FORTRAN_WRAPPER(stpsv)
extern void stpsv(
    char   *uplo,
    char   *trans,
    char   *diag,
    ptrdiff_t *n,
    float  *ap,
    float  *x,
    ptrdiff_t *incx
);

/* Source: strmm.f */
#define strmm FORTRAN_WRAPPER(strmm)
extern void strmm(
    char   *side,
    char   *uplo,
    char   *transa,
    char   *diag,
    ptrdiff_t *m,
    ptrdiff_t *n,
    float  *alpha,
    float  *a,
    ptrdiff_t *lda,
    float  *b,
    ptrdiff_t *ldb
);

/* Source: strmv.f */
#define strmv FORTRAN_WRAPPER(strmv)
extern void strmv(
    char   *uplo,
    char   *trans,
    char   *diag,
    ptrdiff_t *n,
    float  *a,
    ptrdiff_t *lda,
    float  *x,
    ptrdiff_t *incx
);

/* Source: strsm.f */
#define strsm FORTRAN_WRAPPER(strsm)
extern void strsm(
    char   *side,
    char   *uplo,
    char   *transa,
    char   *diag,
    ptrdiff_t *m,
    ptrdiff_t *n,
    float  *alpha,
    float  *a,
    ptrdiff_t *lda,
    float  *b,
    ptrdiff_t *ldb
);

/* Source: strsv.f */
#define strsv FORTRAN_WRAPPER(strsv)
extern void strsv(
    char   *uplo,
    char   *trans,
    char   *diag,
    ptrdiff_t *n,
    float  *a,
    ptrdiff_t *lda,
    float  *x,
    ptrdiff_t *incx
);

/* Source: xerbla.f */
#define xerbla FORTRAN_WRAPPER(xerbla)
extern void xerbla(
    char   *srname,
    ptrdiff_t *info
);

/* Source: zaxpy.f */
#define zaxpy FORTRAN_WRAPPER(zaxpy)
extern void zaxpy(
    ptrdiff_t *n,
    double *za,
    double *zx,
    ptrdiff_t *incx,
    double *zy,
    ptrdiff_t *incy
);

/* Source: zcopy.f */
#define zcopy FORTRAN_WRAPPER(zcopy)
extern void zcopy(
    ptrdiff_t *n,
    double *zx,
    ptrdiff_t *incx,
    double *zy,
    ptrdiff_t *incy
);

/* Source: zdotc.f */
#define zdotc FORTRAN_WRAPPER(zdotc)
#ifndef FORTRAN_COMPLEX_FUNCTIONS_RETURN_VOID
extern doublecomplex zdotc(
#else
extern void zdotc(
    doublecomplex* retval,
#endif
    ptrdiff_t *n,
    double *zx,
    ptrdiff_t *incx,
    double *zy,
    ptrdiff_t *incy
);

/* Source: zdotu.f */
#define zdotu FORTRAN_WRAPPER(zdotu)
#ifndef FORTRAN_COMPLEX_FUNCTIONS_RETURN_VOID
extern doublecomplex zdotu(
#else
extern void zdotu(
    doublecomplex* retval,
#endif
    ptrdiff_t *n,
    double *zx,
    ptrdiff_t *incx,
    double *zy,
    ptrdiff_t *incy
);

/* Source: zdrot.f */
#define zdrot FORTRAN_WRAPPER(zdrot)
extern void zdrot(
    ptrdiff_t *n,
    double *cx,
    ptrdiff_t *incx,
    double *cy,
    ptrdiff_t *incy,
    double *c,
    double *s
);

/* Source: zdscal.f */
#define zdscal FORTRAN_WRAPPER(zdscal)
extern void zdscal(
    ptrdiff_t *n,
    double *da,
    double *zx,
    ptrdiff_t *incx
);

/* Source: zgbmv.f */
#define zgbmv FORTRAN_WRAPPER(zgbmv)
extern void zgbmv(
    char   *trans,
    ptrdiff_t *m,
    ptrdiff_t *n,
    ptrdiff_t *kl,
    ptrdiff_t *ku,
    double *alpha,
    double *a,
    ptrdiff_t *lda,
    double *x,
    ptrdiff_t *incx,
    double *beta,
    double *y,
    ptrdiff_t *incy
);

/* Source: zgemm.f */
#define zgemm FORTRAN_WRAPPER(zgemm)
extern void zgemm(
    char   *transa,
    char   *transb,
    ptrdiff_t *m,
    ptrdiff_t *n,
    ptrdiff_t *k,
    double *alpha,
    double *a,
    ptrdiff_t *lda,
    double *b,
    ptrdiff_t *ldb,
    double *beta,
    double *c,
    ptrdiff_t *ldc
);

/* Source: zgemv.f */
#define zgemv FORTRAN_WRAPPER(zgemv)
extern void zgemv(
    char   *trans,
    ptrdiff_t *m,
    ptrdiff_t *n,
    double *alpha,
    double *a,
    ptrdiff_t *lda,
    double *x,
    ptrdiff_t *incx,
    double *beta,
    double *y,
    ptrdiff_t *incy
);

/* Source: zgerc.f */
#define zgerc FORTRAN_WRAPPER(zgerc)
extern void zgerc(
    ptrdiff_t *m,
    ptrdiff_t *n,
    double *alpha,
    double *x,
    ptrdiff_t *incx,
    double *y,
    ptrdiff_t *incy,
    double *a,
    ptrdiff_t *lda
);

/* Source: zgeru.f */
#define zgeru FORTRAN_WRAPPER(zgeru)
extern void zgeru(
    ptrdiff_t *m,
    ptrdiff_t *n,
    double *alpha,
    double *x,
    ptrdiff_t *incx,
    double *y,
    ptrdiff_t *incy,
    double *a,
    ptrdiff_t *lda
);

/* Source: zhbmv.f */
#define zhbmv FORTRAN_WRAPPER(zhbmv)
extern void zhbmv(
    char   *uplo,
    ptrdiff_t *n,
    ptrdiff_t *k,
    double *alpha,
    double *a,
    ptrdiff_t *lda,
    double *x,
    ptrdiff_t *incx,
    double *beta,
    double *y,
    ptrdiff_t *incy
);

/* Source: zhemm.f */
#define zhemm FORTRAN_WRAPPER(zhemm)
extern void zhemm(
    char   *side,
    char   *uplo,
    ptrdiff_t *m,
    ptrdiff_t *n,
    double *alpha,
    double *a,
    ptrdiff_t *lda,
    double *b,
    ptrdiff_t *ldb,
    double *beta,
    double *c,
    ptrdiff_t *ldc
);

/* Source: zhemv.f */
#define zhemv FORTRAN_WRAPPER(zhemv)
extern void zhemv(
    char   *uplo,
    ptrdiff_t *n,
    double *alpha,
    double *a,
    ptrdiff_t *lda,
    double *x,
    ptrdiff_t *incx,
    double *beta,
    double *y,
    ptrdiff_t *incy
);

/* Source: zher.f */
#define zher FORTRAN_WRAPPER(zher)
extern void zher(
    char   *uplo,
    ptrdiff_t *n,
    double *alpha,
    double *x,
    ptrdiff_t *incx,
    double *a,
    ptrdiff_t *lda
);

/* Source: zher2.f */
#define zher2 FORTRAN_WRAPPER(zher2)
extern void zher2(
    char   *uplo,
    ptrdiff_t *n,
    double *alpha,
    double *x,
    ptrdiff_t *incx,
    double *y,
    ptrdiff_t *incy,
    double *a,
    ptrdiff_t *lda
);

/* Source: zher2k.f */
#define zher2k FORTRAN_WRAPPER(zher2k)
extern void zher2k(
    char   *uplo,
    char   *trans,
    ptrdiff_t *n,
    ptrdiff_t *k,
    double *alpha,
    double *a,
    ptrdiff_t *lda,
    double *b,
    ptrdiff_t *ldb,
    double *beta,
    double *c,
    ptrdiff_t *ldc
);

/* Source: zherk.f */
#define zherk FORTRAN_WRAPPER(zherk)
extern void zherk(
    char   *uplo,
    char   *trans,
    ptrdiff_t *n,
    ptrdiff_t *k,
    double *alpha,
    double *a,
    ptrdiff_t *lda,
    double *beta,
    double *c,
    ptrdiff_t *ldc
);

/* Source: zhpmv.f */
#define zhpmv FORTRAN_WRAPPER(zhpmv)
extern void zhpmv(
    char   *uplo,
    ptrdiff_t *n,
    double *alpha,
    double *ap,
    double *x,
    ptrdiff_t *incx,
    double *beta,
    double *y,
    ptrdiff_t *incy
);

/* Source: zhpr.f */
#define zhpr FORTRAN_WRAPPER(zhpr)
extern void zhpr(
    char   *uplo,
    ptrdiff_t *n,
    double *alpha,
    double *x,
    ptrdiff_t *incx,
    double *ap
);

/* Source: zhpr2.f */
#define zhpr2 FORTRAN_WRAPPER(zhpr2)
extern void zhpr2(
    char   *uplo,
    ptrdiff_t *n,
    double *alpha,
    double *x,
    ptrdiff_t *incx,
    double *y,
    ptrdiff_t *incy,
    double *ap
);

/* Source: zrotg.f */
#define zrotg FORTRAN_WRAPPER(zrotg)
extern void zrotg(
    double *ca,
    double *cb,
    double *c,
    double *s
);

/* Source: zscal.f */
#define zscal FORTRAN_WRAPPER(zscal)
extern void zscal(
    ptrdiff_t *n,
    double *za,
    double *zx,
    ptrdiff_t *incx
);

/* Source: zswap.f */
#define zswap FORTRAN_WRAPPER(zswap)
extern void zswap(
    ptrdiff_t *n,
    double *zx,
    ptrdiff_t *incx,
    double *zy,
    ptrdiff_t *incy
);

/* Source: zsymm.f */
#define zsymm FORTRAN_WRAPPER(zsymm)
extern void zsymm(
    char   *side,
    char   *uplo,
    ptrdiff_t *m,
    ptrdiff_t *n,
    double *alpha,
    double *a,
    ptrdiff_t *lda,
    double *b,
    ptrdiff_t *ldb,
    double *beta,
    double *c,
    ptrdiff_t *ldc
);

/* Source: zsyr2k.f */
#define zsyr2k FORTRAN_WRAPPER(zsyr2k)
extern void zsyr2k(
    char   *uplo,
    char   *trans,
    ptrdiff_t *n,
    ptrdiff_t *k,
    double *alpha,
    double *a,
    ptrdiff_t *lda,
    double *b,
    ptrdiff_t *ldb,
    double *beta,
    double *c,
    ptrdiff_t *ldc
);

/* Source: zsyrk.f */
#define zsyrk FORTRAN_WRAPPER(zsyrk)
extern void zsyrk(
    char   *uplo,
    char   *trans,
    ptrdiff_t *n,
    ptrdiff_t *k,
    double *alpha,
    double *a,
    ptrdiff_t *lda,
    double *beta,
    double *c,
    ptrdiff_t *ldc
);

/* Source: ztbmv.f */
#define ztbmv FORTRAN_WRAPPER(ztbmv)
extern void ztbmv(
    char   *uplo,
    char   *trans,
    char   *diag,
    ptrdiff_t *n,
    ptrdiff_t *k,
    double *a,
    ptrdiff_t *lda,
    double *x,
    ptrdiff_t *incx
);

/* Source: ztbsv.f */
#define ztbsv FORTRAN_WRAPPER(ztbsv)
extern void ztbsv(
    char   *uplo,
    char   *trans,
    char   *diag,
    ptrdiff_t *n,
    ptrdiff_t *k,
    double *a,
    ptrdiff_t *lda,
    double *x,
    ptrdiff_t *incx
);

/* Source: ztpmv.f */
#define ztpmv FORTRAN_WRAPPER(ztpmv)
extern void ztpmv(
    char   *uplo,
    char   *trans,
    char   *diag,
    ptrdiff_t *n,
    double *ap,
    double *x,
    ptrdiff_t *incx
);

/* Source: ztpsv.f */
#define ztpsv FORTRAN_WRAPPER(ztpsv)
extern void ztpsv(
    char   *uplo,
    char   *trans,
    char   *diag,
    ptrdiff_t *n,
    double *ap,
    double *x,
    ptrdiff_t *incx
);

/* Source: ztrmm.f */
#define ztrmm FORTRAN_WRAPPER(ztrmm)
extern void ztrmm(
    char   *side,
    char   *uplo,
    char   *transa,
    char   *diag,
    ptrdiff_t *m,
    ptrdiff_t *n,
    double *alpha,
    double *a,
    ptrdiff_t *lda,
    double *b,
    ptrdiff_t *ldb
);

/* Source: ztrmv.f */
#define ztrmv FORTRAN_WRAPPER(ztrmv)
extern void ztrmv(
    char   *uplo,
    char   *trans,
    char   *diag,
    ptrdiff_t *n,
    double *a,
    ptrdiff_t *lda,
    double *x,
    ptrdiff_t *incx
);

/* Source: ztrsm.f */
#define ztrsm FORTRAN_WRAPPER(ztrsm)
extern void ztrsm(
    char   *side,
    char   *uplo,
    char   *transa,
    char   *diag,
    ptrdiff_t *m,
    ptrdiff_t *n,
    double *alpha,
    double *a,
    ptrdiff_t *lda,
    double *b,
    ptrdiff_t *ldb
);

/* Source: ztrsv.f */
#define ztrsv FORTRAN_WRAPPER(ztrsv)
extern void ztrsv(
    char   *uplo,
    char   *trans,
    char   *diag,
    ptrdiff_t *n,
    double *a,
    ptrdiff_t *lda,
    double *x,
    ptrdiff_t *incx
);

#ifdef __cplusplus
    }   /* extern "C" */
#endif

#endif /* blas_h */
```
